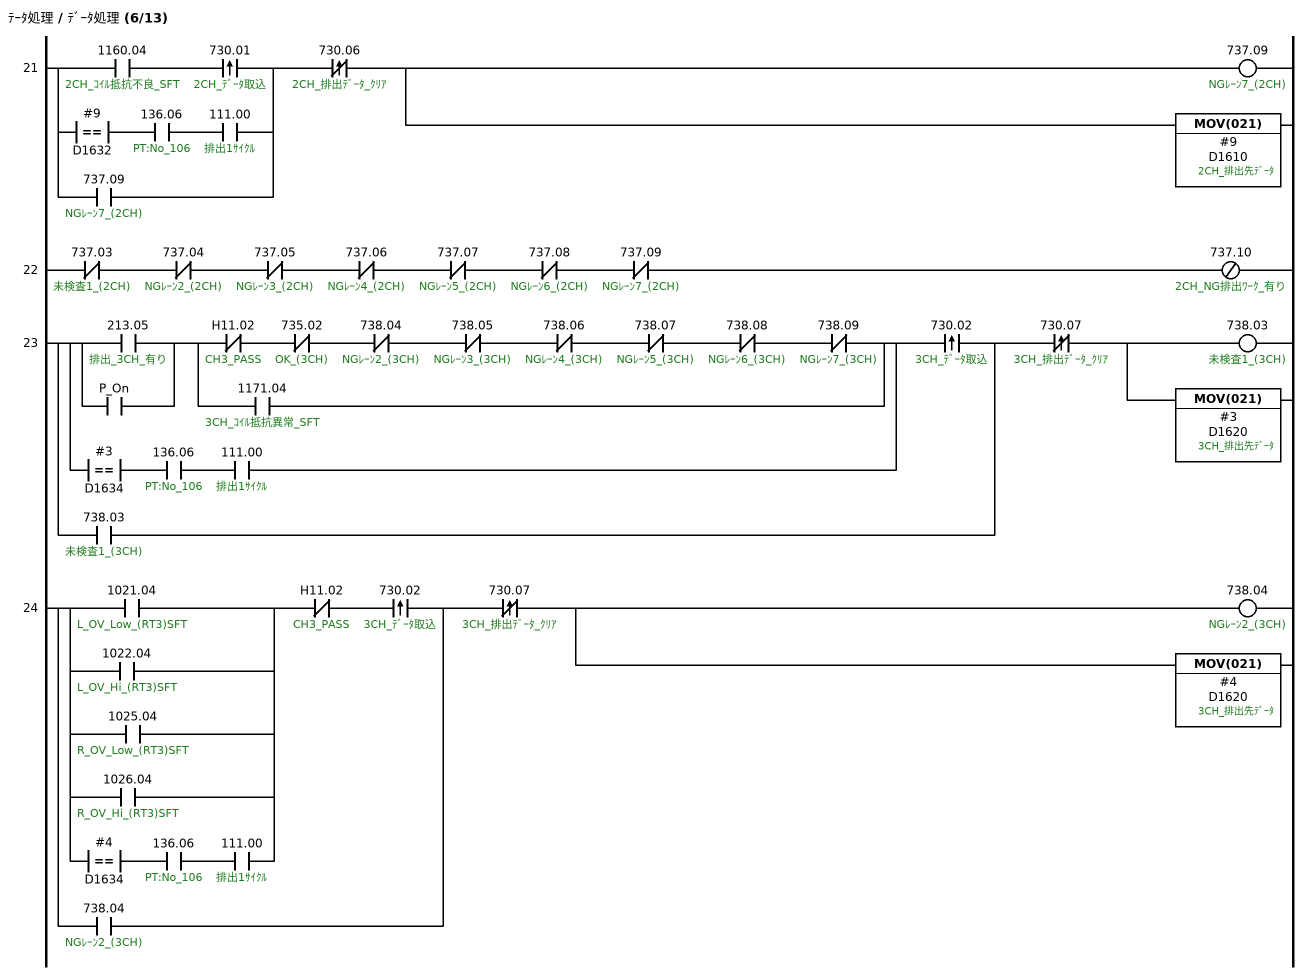
; [picture p168: ﾃｰﾀ処理 / ﾃﾞｰﾀ処理, rungs 21-24]
; rung 21
LD 1160.04  ; 2CH_ｺｲﾙ抵抗不良_SFT
@AND 730.01  ; 2CH_ﾃﾞｰﾀ取込
LD=(300) #9 D1632
AND 136.06  ; PT:No_106
AND 111.00  ; 排出1ｻｲｸﾙ
ORLD
OR 737.09  ; NGﾚｰﾝ7_(2CH)
@ANDNOT 730.06  ; 2CH_排出ﾃﾞｰﾀ_ｸﾘｱ
OUT 737.09  ; NGﾚｰﾝ7_(2CH)
MOV(021) #9 D1610  ; 2CH_排出先ﾃﾞｰﾀ
; rung 22
LDNOT 737.03  ; 未検査1_(2CH)
ANDNOT 737.04  ; NGﾚｰﾝ2_(2CH)
ANDNOT 737.05  ; NGﾚｰﾝ3_(2CH)
ANDNOT 737.06  ; NGﾚｰﾝ4_(2CH)
ANDNOT 737.07  ; NGﾚｰﾝ5_(2CH)
ANDNOT 737.08  ; NGﾚｰﾝ6_(2CH)
ANDNOT 737.09  ; NGﾚｰﾝ7_(2CH)
OUTNOT 737.10  ; 2CH_NG排出ﾜｰｸ_有り
; rung 23
LD 213.05  ; 排出_3CH_有り
OR P_On
LDNOT H11.02  ; CH3_PASS
ANDNOT 735.02  ; OK_(3CH)
ANDNOT 738.04  ; NGﾚｰﾝ2_(3CH)
ANDNOT 738.05  ; NGﾚｰﾝ3_(3CH)
ANDNOT 738.06  ; NGﾚｰﾝ4_(3CH)
ANDNOT 738.07  ; NGﾚｰﾝ5_(3CH)
ANDNOT 738.08  ; NGﾚｰﾝ6_(3CH)
ANDNOT 738.09  ; NGﾚｰﾝ7_(3CH)
OR 1171.04  ; 3CH_ｺｲﾙ抵抗異常_SFT
ANDLD
LD=(300) #3 D1634
AND 136.06  ; PT:No_106
AND 111.00  ; 排出1ｻｲｸﾙ
ORLD
@AND 730.02  ; 3CH_ﾃﾞｰﾀ取込
OR 738.03  ; 未検査1_(3CH)
@ANDNOT 730.07  ; 3CH_排出ﾃﾞｰﾀ_ｸﾘｱ
OUT 738.03  ; 未検査1_(3CH)
MOV(021) #3 D1620  ; 3CH_排出先ﾃﾞｰﾀ
; rung 24
LD 1021.04  ; L_OV_Low_(RT3)SFT
OR 1022.04  ; L_OV_Hi_(RT3)SFT
OR 1025.04  ; R_OV_Low_(RT3)SFT
OR 1026.04  ; R_OV_Hi_(RT3)SFT
LD=(300) #4 D1634
AND 136.06  ; PT:No_106
AND 111.00  ; 排出1ｻｲｸﾙ
ORLD
ANDNOT H11.02  ; CH3_PASS
@AND 730.02  ; 3CH_ﾃﾞｰﾀ取込
OR 738.04  ; NGﾚｰﾝ2_(3CH)
@ANDNOT 730.07  ; 3CH_排出ﾃﾞｰﾀ_ｸﾘｱ
OUT 738.04  ; NGﾚｰﾝ2_(3CH)
MOV(021) #4 D1620  ; 3CH_排出先ﾃﾞｰﾀ

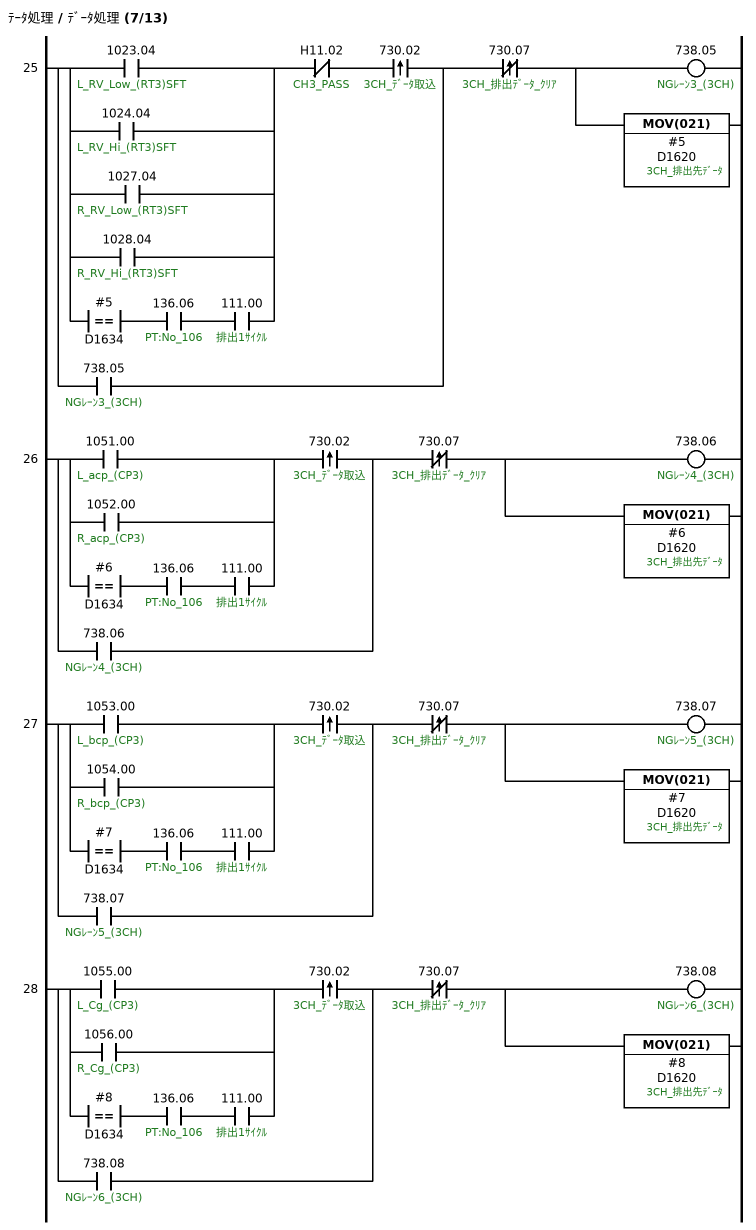
; rung 25
LD 1023.04  ; L_RV_Low_(RT3)SFT
OR 1024.04  ; L_RV_Hi_(RT3)SFT
OR 1027.04  ; R_RV_Low_(RT3)SFT
OR 1028.04  ; R_RV_Hi_(RT3)SFT
LD=(300) #5 D1634
AND 136.06  ; PT:No_106
AND 111.00  ; 排出1ｻｲｸﾙ
ORLD
ANDNOT H11.02  ; CH3_PASS
@AND 730.02  ; 3CH_ﾃﾞｰﾀ取込
OR 738.05  ; NGﾚｰﾝ3_(3CH)
@ANDNOT 730.07  ; 3CH_排出ﾃﾞｰﾀ_ｸﾘｱ
OUT 738.05  ; NGﾚｰﾝ3_(3CH)
MOV(021) #5 D1620  ; 3CH_排出先ﾃﾞｰﾀ
; rung 26
LD 1051.00  ; L_acp_(CP3)
OR 1052.00  ; R_acp_(CP3)
LD=(300) #6 D1634
AND 136.06  ; PT:No_106
AND 111.00  ; 排出1ｻｲｸﾙ
ORLD
@AND 730.02  ; 3CH_ﾃﾞｰﾀ取込
OR 738.06  ; NGﾚｰﾝ4_(3CH)
@ANDNOT 730.07  ; 3CH_排出ﾃﾞｰﾀ_ｸﾘｱ
OUT 738.06  ; NGﾚｰﾝ4_(3CH)
MOV(021) #6 D1620  ; 3CH_排出先ﾃﾞｰﾀ
; rung 27
LD 1053.00  ; L_bcp_(CP3)
OR 1054.00  ; R_bcp_(CP3)
LD=(300) #7 D1634
AND 136.06  ; PT:No_106
AND 111.00  ; 排出1ｻｲｸﾙ
ORLD
@AND 730.02  ; 3CH_ﾃﾞｰﾀ取込
OR 738.07  ; NGﾚｰﾝ5_(3CH)
@ANDNOT 730.07  ; 3CH_排出ﾃﾞｰﾀ_ｸﾘｱ
OUT 738.07  ; NGﾚｰﾝ5_(3CH)
MOV(021) #7 D1620  ; 3CH_排出先ﾃﾞｰﾀ
; rung 28
LD 1055.00  ; L_Cg_(CP3)
OR 1056.00  ; R_Cg_(CP3)
LD=(300) #8 D1634
AND 136.06  ; PT:No_106
AND 111.00  ; 排出1ｻｲｸﾙ
ORLD
@AND 730.02  ; 3CH_ﾃﾞｰﾀ取込
OR 738.08  ; NGﾚｰﾝ6_(3CH)
@ANDNOT 730.07  ; 3CH_排出ﾃﾞｰﾀ_ｸﾘｱ
OUT 738.08  ; NGﾚｰﾝ6_(3CH)
MOV(021) #8 D1620  ; 3CH_排出先ﾃﾞｰﾀ

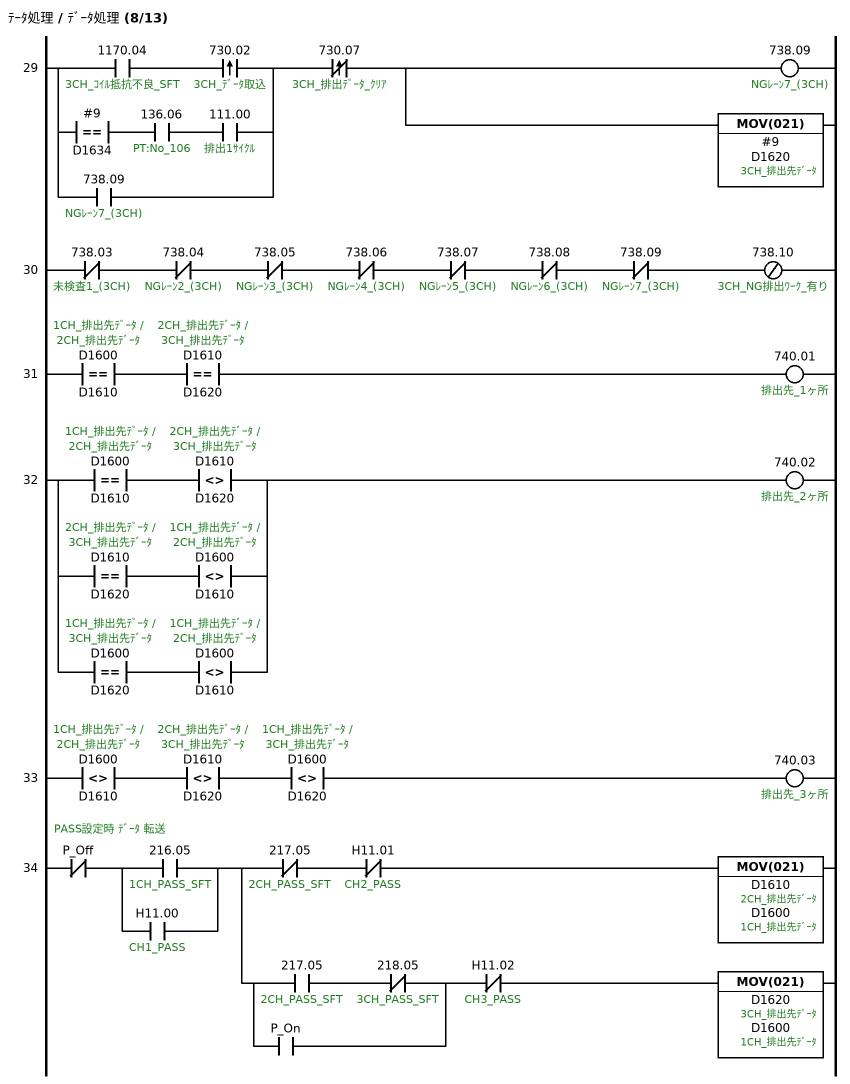
; rung 29
LD 1170.04  ; 3CH_ｺｲﾙ抵抗不良_SFT
@AND 730.02  ; 3CH_ﾃﾞｰﾀ取込
LD=(300) #9 D1634
AND 136.06  ; PT:No_106
AND 111.00  ; 排出1ｻｲｸﾙ
ORLD
OR 738.09  ; NGﾚｰﾝ7_(3CH)
@ANDNOT 730.07  ; 3CH_排出ﾃﾞｰﾀ_ｸﾘｱ
OUT 738.09  ; NGﾚｰﾝ7_(3CH)
MOV(021) #9 D1620  ; 3CH_排出先ﾃﾞｰﾀ
; rung 30
LDNOT 738.03  ; 未検査1_(3CH)
ANDNOT 738.04  ; NGﾚｰﾝ2_(3CH)
ANDNOT 738.05  ; NGﾚｰﾝ3_(3CH)
ANDNOT 738.06  ; NGﾚｰﾝ4_(3CH)
ANDNOT 738.07  ; NGﾚｰﾝ5_(3CH)
ANDNOT 738.08  ; NGﾚｰﾝ6_(3CH)
ANDNOT 738.09  ; NGﾚｰﾝ7_(3CH)
OUTNOT 738.10  ; 3CH_NG排出ﾜｰｸ_有り
; rung 31
LD=(300) D1600 D1610  ; 1CH_排出先ﾃﾞｰﾀ, 2CH_排出先ﾃﾞｰﾀ
AND=(300) D1610 D1620  ; 2CH_排出先ﾃﾞｰﾀ, 3CH_排出先ﾃﾞｰﾀ
OUT 740.01  ; 排出先_1ヶ所
; rung 32
LD=(300) D1600 D1610  ; 1CH_排出先ﾃﾞｰﾀ, 2CH_排出先ﾃﾞｰﾀ
AND<>(305) D1610 D1620  ; 2CH_排出先ﾃﾞｰﾀ, 3CH_排出先ﾃﾞｰﾀ
LD=(300) D1610 D1620  ; 2CH_排出先ﾃﾞｰﾀ, 3CH_排出先ﾃﾞｰﾀ
AND<>(305) D1600 D1610  ; 1CH_排出先ﾃﾞｰﾀ, 2CH_排出先ﾃﾞｰﾀ
ORLD
LD=(300) D1600 D1620  ; 1CH_排出先ﾃﾞｰﾀ, 3CH_排出先ﾃﾞｰﾀ
AND<>(305) D1600 D1610  ; 1CH_排出先ﾃﾞｰﾀ, 2CH_排出先ﾃﾞｰﾀ
ORLD
OUT 740.02  ; 排出先_2ヶ所
; rung 33
LD<>(305) D1600 D1610  ; 1CH_排出先ﾃﾞｰﾀ, 2CH_排出先ﾃﾞｰﾀ
AND<>(305) D1610 D1620  ; 2CH_排出先ﾃﾞｰﾀ, 3CH_排出先ﾃﾞｰﾀ
AND<>(305) D1600 D1620  ; 1CH_排出先ﾃﾞｰﾀ, 3CH_排出先ﾃﾞｰﾀ
OUT 740.03  ; 排出先_3ヶ所
; rung 34: PASS設定時 ﾃﾞｰﾀ 転送
LDNOT P_Off
LD 216.05  ; 1CH_PASS_SFT
OR H11.00  ; CH1_PASS
ANDLD
OUT TR0
ANDNOT 217.05  ; 2CH_PASS_SFT
ANDNOT H11.01  ; CH2_PASS
MOV(021) D1610 D1600  ; 2CH_排出先ﾃﾞｰﾀ, 1CH_排出先ﾃﾞｰﾀ
LD TR0
LD 217.05  ; 2CH_PASS_SFT
ANDNOT 218.05  ; 3CH_PASS_SFT
OR P_On
ANDLD
ANDNOT H11.02  ; CH3_PASS
MOV(021) D1620 D1600  ; 3CH_排出先ﾃﾞｰﾀ, 1CH_排出先ﾃﾞｰﾀ

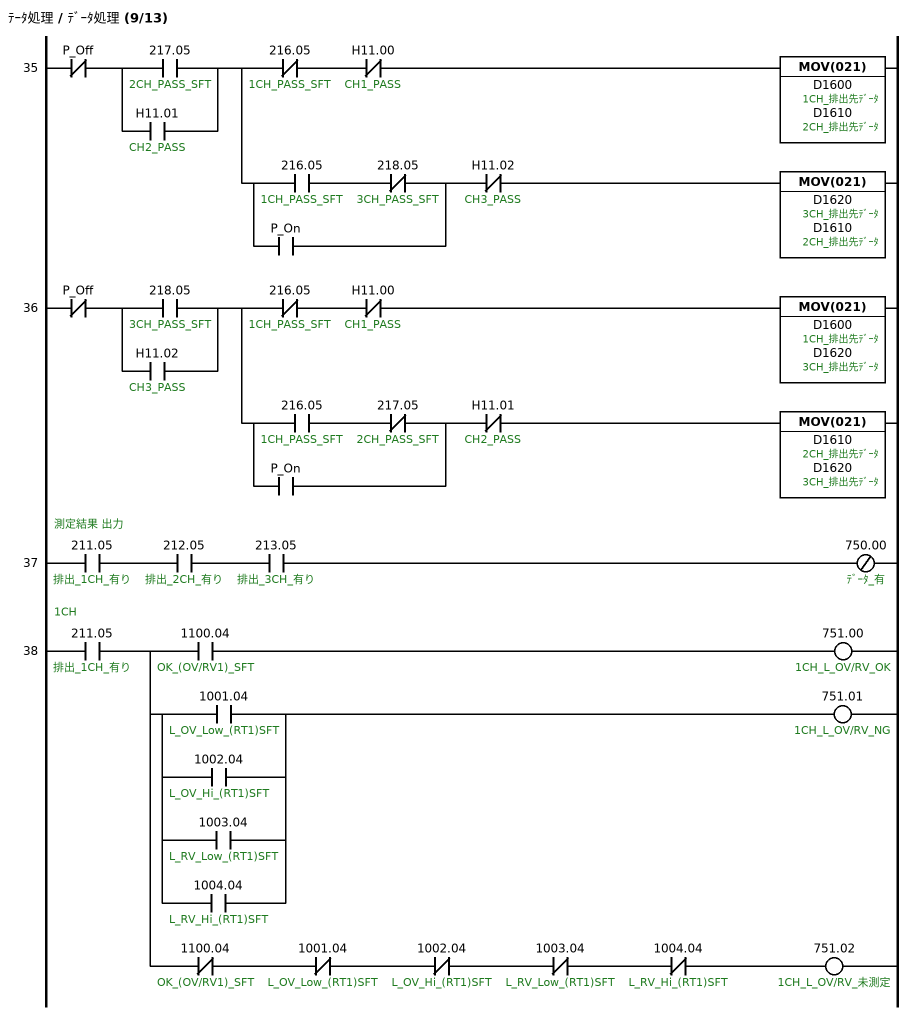
; rung 35
LDNOT P_Off
LD 217.05  ; 2CH_PASS_SFT
OR H11.01  ; CH2_PASS
ANDLD
OUT TR0
ANDNOT 216.05  ; 1CH_PASS_SFT
ANDNOT H11.00  ; CH1_PASS
MOV(021) D1600 D1610  ; 1CH_排出先ﾃﾞｰﾀ, 2CH_排出先ﾃﾞｰﾀ
LD TR0
LD 216.05  ; 1CH_PASS_SFT
ANDNOT 218.05  ; 3CH_PASS_SFT
OR P_On
ANDLD
ANDNOT H11.02  ; CH3_PASS
MOV(021) D1620 D1610  ; 3CH_排出先ﾃﾞｰﾀ, 2CH_排出先ﾃﾞｰﾀ
; rung 36
LDNOT P_Off
LD 218.05  ; 3CH_PASS_SFT
OR H11.02  ; CH3_PASS
ANDLD
OUT TR0
ANDNOT 216.05  ; 1CH_PASS_SFT
ANDNOT H11.00  ; CH1_PASS
MOV(021) D1600 D1620  ; 1CH_排出先ﾃﾞｰﾀ, 3CH_排出先ﾃﾞｰﾀ
LD TR0
LD 216.05  ; 1CH_PASS_SFT
ANDNOT 217.05  ; 2CH_PASS_SFT
OR P_On
ANDLD
ANDNOT H11.01  ; CH2_PASS
MOV(021) D1610 D1620  ; 2CH_排出先ﾃﾞｰﾀ, 3CH_排出先ﾃﾞｰﾀ
; rung 37: 測定結果 出力
LD 211.05  ; 排出_1CH_有り
AND 212.05  ; 排出_2CH_有り
AND 213.05  ; 排出_3CH_有り
OUTNOT 750.00  ; ﾃﾞｰﾀ_有
; rung 38: 1CH
LD 211.05  ; 排出_1CH_有り
OUT TR0
AND 1100.04  ; OK_(OV/RV1)_SFT
OUT 751.00  ; 1CH_L_OV/RV_OK
LD TR0
LD 1001.04  ; L_OV_Low_(RT1)SFT
OR 1002.04  ; L_OV_Hi_(RT1)SFT
OR 1003.04  ; L_RV_Low_(RT1)SFT
OR 1004.04  ; L_RV_Hi_(RT1)SFT
ANDLD
OUT 751.01  ; 1CH_L_OV/RV_NG
LD TR0
ANDNOT 1100.04  ; OK_(OV/RV1)_SFT
ANDNOT 1001.04  ; L_OV_Low_(RT1)SFT
ANDNOT 1002.04  ; L_OV_Hi_(RT1)SFT
ANDNOT 1003.04  ; L_RV_Low_(RT1)SFT
ANDNOT 1004.04  ; L_RV_Hi_(RT1)SFT
OUT 751.02  ; 1CH_L_OV/RV_未測定

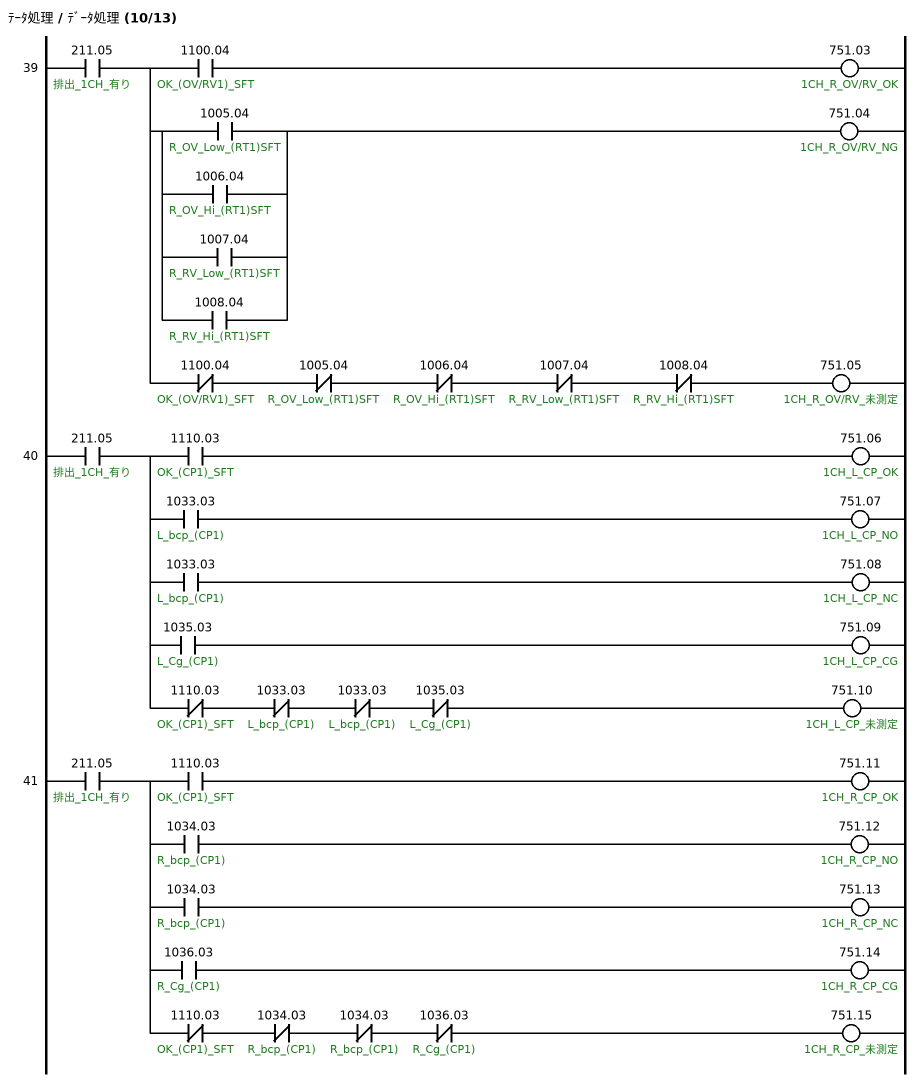
; rung 39
LD 211.05  ; 排出_1CH_有り
OUT TR0
AND 1100.04  ; OK_(OV/RV1)_SFT
OUT 751.03  ; 1CH_R_OV/RV_OK
LD TR0
LD 1005.04  ; R_OV_Low_(RT1)SFT
OR 1006.04  ; R_OV_Hi_(RT1)SFT
OR 1007.04  ; R_RV_Low_(RT1)SFT
OR 1008.04  ; R_RV_Hi_(RT1)SFT
ANDLD
OUT 751.04  ; 1CH_R_OV/RV_NG
LD TR0
ANDNOT 1100.04  ; OK_(OV/RV1)_SFT
ANDNOT 1005.04  ; R_OV_Low_(RT1)SFT
ANDNOT 1006.04  ; R_OV_Hi_(RT1)SFT
ANDNOT 1007.04  ; R_RV_Low_(RT1)SFT
ANDNOT 1008.04  ; R_RV_Hi_(RT1)SFT
OUT 751.05  ; 1CH_R_OV/RV_未測定
; rung 40
LD 211.05  ; 排出_1CH_有り
OUT TR0
AND 1110.03  ; OK_(CP1)_SFT
OUT 751.06  ; 1CH_L_CP_OK
LD TR0
AND 1033.03  ; L_bcp_(CP1)
OUT 751.07  ; 1CH_L_CP_NO
LD TR0
AND 1033.03  ; L_bcp_(CP1)
OUT 751.08  ; 1CH_L_CP_NC
LD TR0
AND 1035.03  ; L_Cg_(CP1)
OUT 751.09  ; 1CH_L_CP_CG
LD TR0
ANDNOT 1110.03  ; OK_(CP1)_SFT
ANDNOT 1033.03  ; L_bcp_(CP1)
ANDNOT 1033.03  ; L_bcp_(CP1)
ANDNOT 1035.03  ; L_Cg_(CP1)
OUT 751.10  ; 1CH_L_CP_未測定
; rung 41
LD 211.05  ; 排出_1CH_有り
OUT TR0
AND 1110.03  ; OK_(CP1)_SFT
OUT 751.11  ; 1CH_R_CP_OK
LD TR0
AND 1034.03  ; R_bcp_(CP1)
OUT 751.12  ; 1CH_R_CP_NO
LD TR0
AND 1034.03  ; R_bcp_(CP1)
OUT 751.13  ; 1CH_R_CP_NC
LD TR0
AND 1036.03  ; R_Cg_(CP1)
OUT 751.14  ; 1CH_R_CP_CG
LD TR0
ANDNOT 1110.03  ; OK_(CP1)_SFT
ANDNOT 1034.03  ; R_bcp_(CP1)
ANDNOT 1034.03  ; R_bcp_(CP1)
ANDNOT 1036.03  ; R_Cg_(CP1)
OUT 751.15  ; 1CH_R_CP_未測定

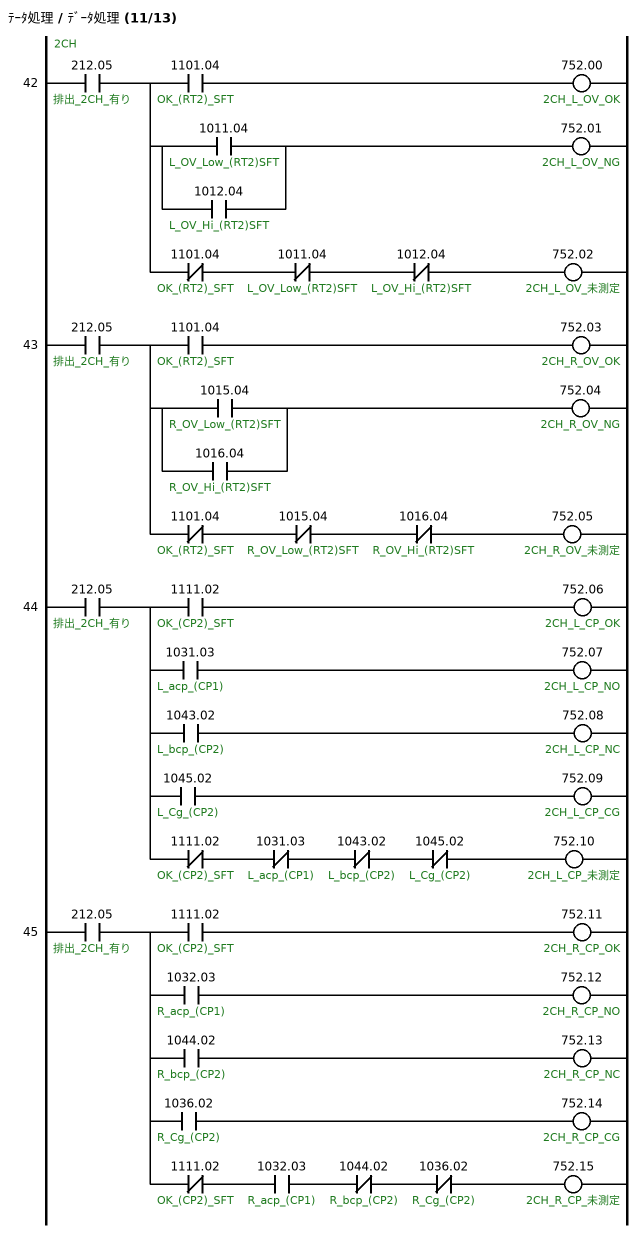
; rung 42: 2CH
LD 212.05  ; 排出_2CH_有り
OUT TR0
AND 1101.04  ; OK_(RT2)_SFT
OUT 752.00  ; 2CH_L_OV_OK
LD TR0
LD 1011.04  ; L_OV_Low_(RT2)SFT
OR 1012.04  ; L_OV_Hi_(RT2)SFT
ANDLD
OUT 752.01  ; 2CH_L_OV_NG
LD TR0
ANDNOT 1101.04  ; OK_(RT2)_SFT
ANDNOT 1011.04  ; L_OV_Low_(RT2)SFT
ANDNOT 1012.04  ; L_OV_Hi_(RT2)SFT
OUT 752.02  ; 2CH_L_OV_未測定
; rung 43
LD 212.05  ; 排出_2CH_有り
OUT TR0
AND 1101.04  ; OK_(RT2)_SFT
OUT 752.03  ; 2CH_R_OV_OK
LD TR0
LD 1015.04  ; R_OV_Low_(RT2)SFT
OR 1016.04  ; R_OV_Hi_(RT2)SFT
ANDLD
OUT 752.04  ; 2CH_R_OV_NG
LD TR0
ANDNOT 1101.04  ; OK_(RT2)_SFT
ANDNOT 1015.04  ; R_OV_Low_(RT2)SFT
ANDNOT 1016.04  ; R_OV_Hi_(RT2)SFT
OUT 752.05  ; 2CH_R_OV_未測定
; rung 44
LD 212.05  ; 排出_2CH_有り
OUT TR0
AND 1111.02  ; OK_(CP2)_SFT
OUT 752.06  ; 2CH_L_CP_OK
LD TR0
AND 1031.03  ; L_acp_(CP1)
OUT 752.07  ; 2CH_L_CP_NO
LD TR0
AND 1043.02  ; L_bcp_(CP2)
OUT 752.08  ; 2CH_L_CP_NC
LD TR0
AND 1045.02  ; L_Cg_(CP2)
OUT 752.09  ; 2CH_L_CP_CG
LD TR0
ANDNOT 1111.02  ; OK_(CP2)_SFT
ANDNOT 1031.03  ; L_acp_(CP1)
ANDNOT 1043.02  ; L_bcp_(CP2)
ANDNOT 1045.02  ; L_Cg_(CP2)
OUT 752.10  ; 2CH_L_CP_未測定
; rung 45
LD 212.05  ; 排出_2CH_有り
OUT TR0
AND 1111.02  ; OK_(CP2)_SFT
OUT 752.11  ; 2CH_R_CP_OK
LD TR0
AND 1032.03  ; R_acp_(CP1)
OUT 752.12  ; 2CH_R_CP_NO
LD TR0
AND 1044.02  ; R_bcp_(CP2)
OUT 752.13  ; 2CH_R_CP_NC
LD TR0
AND 1036.02  ; R_Cg_(CP2)
OUT 752.14  ; 2CH_R_CP_CG
LD TR0
ANDNOT 1111.02  ; OK_(CP2)_SFT
AND 1032.03  ; R_acp_(CP1)
ANDNOT 1044.02  ; R_bcp_(CP2)
ANDNOT 1036.02  ; R_Cg_(CP2)
OUT 752.15  ; 2CH_R_CP_未測定

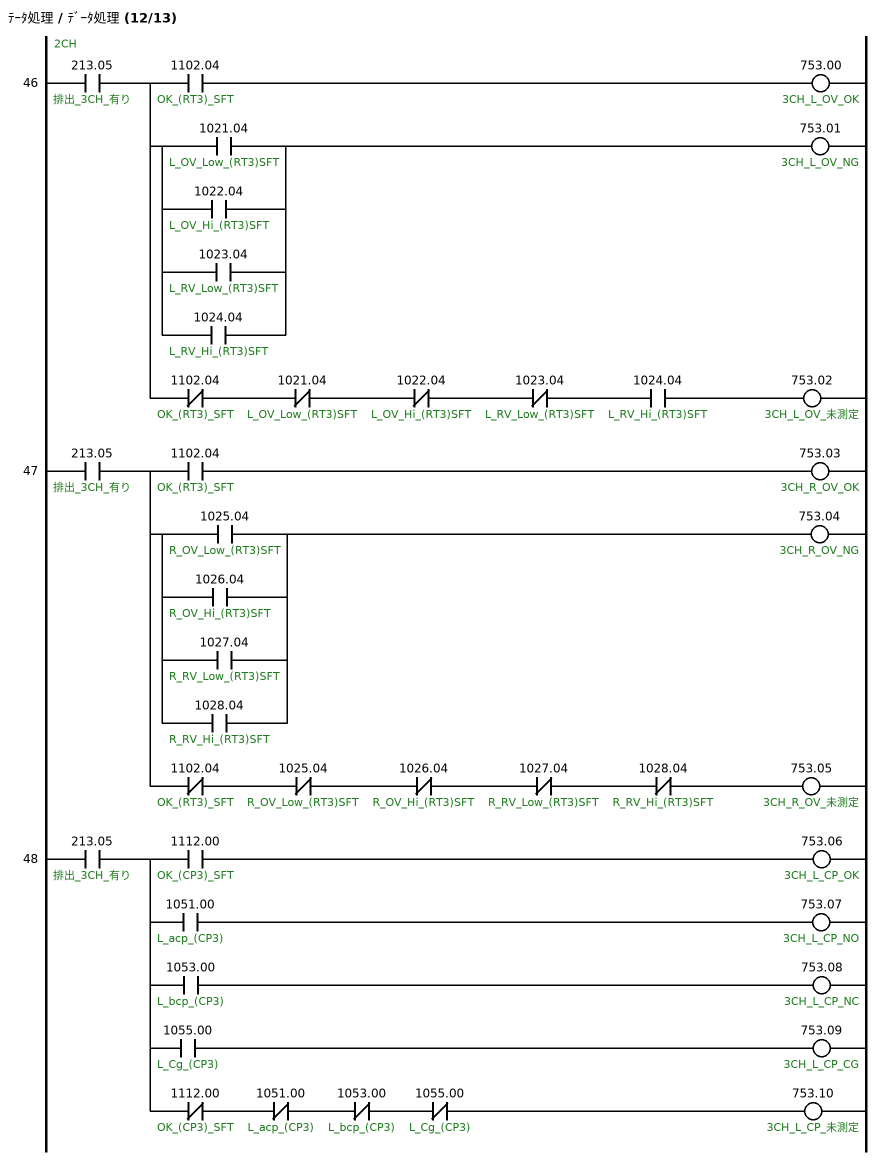
; rung 46: 2CH
LD 213.05  ; 排出_3CH_有り
OUT TR0
AND 1102.04  ; OK_(RT3)_SFT
OUT 753.00  ; 3CH_L_OV_OK
LD TR0
LD 1021.04  ; L_OV_Low_(RT3)SFT
OR 1022.04  ; L_OV_Hi_(RT3)SFT
OR 1023.04  ; L_RV_Low_(RT3)SFT
OR 1024.04  ; L_RV_Hi_(RT3)SFT
ANDLD
OUT 753.01  ; 3CH_L_OV_NG
LD TR0
ANDNOT 1102.04  ; OK_(RT3)_SFT
ANDNOT 1021.04  ; L_OV_Low_(RT3)SFT
ANDNOT 1022.04  ; L_OV_Hi_(RT3)SFT
ANDNOT 1023.04  ; L_RV_Low_(RT3)SFT
AND 1024.04  ; L_RV_Hi_(RT3)SFT
OUT 753.02  ; 3CH_L_OV_未測定
; rung 47
LD 213.05  ; 排出_3CH_有り
OUT TR0
AND 1102.04  ; OK_(RT3)_SFT
OUT 753.03  ; 3CH_R_OV_OK
LD TR0
LD 1025.04  ; R_OV_Low_(RT3)SFT
OR 1026.04  ; R_OV_Hi_(RT3)SFT
OR 1027.04  ; R_RV_Low_(RT3)SFT
OR 1028.04  ; R_RV_Hi_(RT3)SFT
ANDLD
OUT 753.04  ; 3CH_R_OV_NG
LD TR0
ANDNOT 1102.04  ; OK_(RT3)_SFT
ANDNOT 1025.04  ; R_OV_Low_(RT3)SFT
ANDNOT 1026.04  ; R_OV_Hi_(RT3)SFT
ANDNOT 1027.04  ; R_RV_Low_(RT3)SFT
ANDNOT 1028.04  ; R_RV_Hi_(RT3)SFT
OUT 753.05  ; 3CH_R_OV_未測定
; rung 48
LD 213.05  ; 排出_3CH_有り
OUT TR0
AND 1112.00  ; OK_(CP3)_SFT
OUT 753.06  ; 3CH_L_CP_OK
LD TR0
AND 1051.00  ; L_acp_(CP3)
OUT 753.07  ; 3CH_L_CP_NO
LD TR0
AND 1053.00  ; L_bcp_(CP3)
OUT 753.08  ; 3CH_L_CP_NC
LD TR0
AND 1055.00  ; L_Cg_(CP3)
OUT 753.09  ; 3CH_L_CP_CG
LD TR0
ANDNOT 1112.00  ; OK_(CP3)_SFT
ANDNOT 1051.00  ; L_acp_(CP3)
ANDNOT 1053.00  ; L_bcp_(CP3)
ANDNOT 1055.00  ; L_Cg_(CP3)
OUT 753.10  ; 3CH_L_CP_未測定

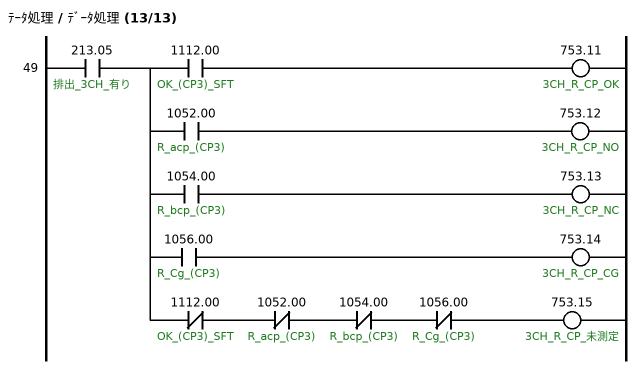
; rung 49
LD 213.05  ; 排出_3CH_有り
OUT TR0
AND 1112.00  ; OK_(CP3)_SFT
OUT 753.11  ; 3CH_R_CP_OK
LD TR0
AND 1052.00  ; R_acp_(CP3)
OUT 753.12  ; 3CH_R_CP_NO
LD TR0
AND 1054.00  ; R_bcp_(CP3)
OUT 753.13  ; 3CH_R_CP_NC
LD TR0
AND 1056.00  ; R_Cg_(CP3)
OUT 753.14  ; 3CH_R_CP_CG
LD TR0
ANDNOT 1112.00  ; OK_(CP3)_SFT
ANDNOT 1052.00  ; R_acp_(CP3)
ANDNOT 1054.00  ; R_bcp_(CP3)
ANDNOT 1056.00  ; R_Cg_(CP3)
OUT 753.15  ; 3CH_R_CP_未測定

### Section END
; rung 0
END(001)

## Program 排出 (cyclic task 7)

### Section 制御

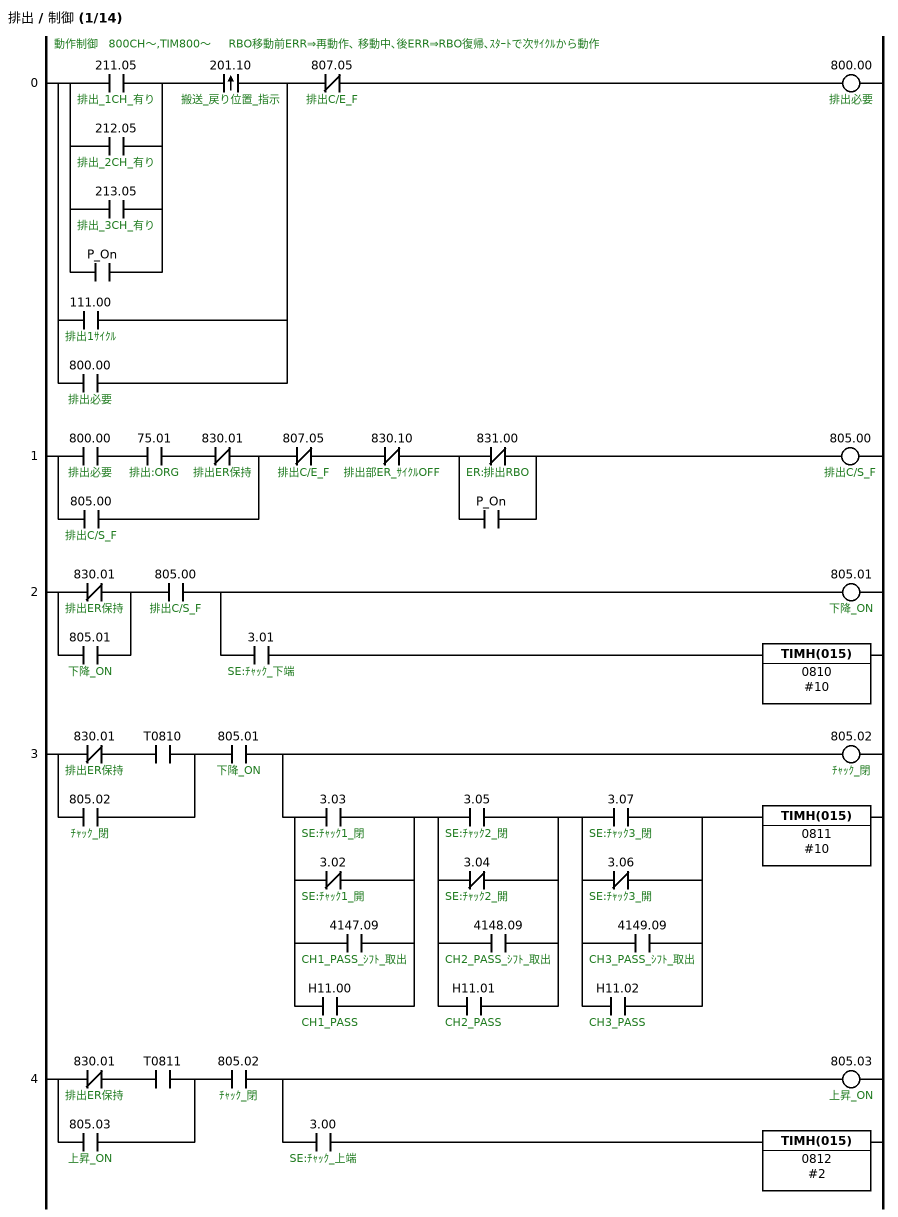
; rung 0: 動作制御   800CH～,TIM800～     RBO移動前ERR⇒再動作､ 移動中､後ERR⇒RBO復帰､ｽﾀｰﾄで次ｻｲｸﾙから動作
LD 211.05  ; 排出_1CH_有り
OR 212.05  ; 排出_2CH_有り
OR 213.05  ; 排出_3CH_有り
OR P_On
@AND 201.10  ; 搬送_戻り位置_指示
OR 111.00  ; 排出1ｻｲｸﾙ
OR 800.00  ; 排出必要
ANDNOT 807.05  ; 排出C/E_F
OUT 800.00  ; 排出必要
; rung 1
LD 800.00  ; 排出必要
AND 75.01  ; 排出:ORG
ANDNOT 830.01  ; 排出ER保持
OR 805.00  ; 排出C/S_F
ANDNOT 807.05  ; 排出C/E_F
ANDNOT 830.10  ; 排出部ER_ｻｲｸﾙOFF
LDNOT 831.00  ; ER:排出RBO
OR P_On
ANDLD
OUT 805.00  ; 排出C/S_F
; rung 2
LDNOT 830.01  ; 排出ER保持
OR 805.01  ; 下降_ON
AND 805.00  ; 排出C/S_F
OUT 805.01  ; 下降_ON
AND 3.01  ; SE:ﾁｬｯｸ_下端
TIMH(015) 0810 #10
; rung 3
LDNOT 830.01  ; 排出ER保持
AND T0810
OR 805.02  ; ﾁｬｯｸ_閉
AND 805.01  ; 下降_ON
OUT 805.02  ; ﾁｬｯｸ_閉
LD 3.03  ; SE:ﾁｬｯｸ1_閉
ORNOT 3.02  ; SE:ﾁｬｯｸ1_開
OR 4147.09  ; CH1_PASS_ｼﾌﾄ_取出
OR H11.00  ; CH1_PASS
ANDLD
LD 3.05  ; SE:ﾁｬｯｸ2_閉
ORNOT 3.04  ; SE:ﾁｬｯｸ2_開
OR 4148.09  ; CH2_PASS_ｼﾌﾄ_取出
OR H11.01  ; CH2_PASS
ANDLD
LD 3.07  ; SE:ﾁｬｯｸ3_閉
ORNOT 3.06  ; SE:ﾁｬｯｸ3_開
OR 4149.09  ; CH3_PASS_ｼﾌﾄ_取出
OR H11.02  ; CH3_PASS
ANDLD
TIMH(015) 0811 #10
; rung 4
LDNOT 830.01  ; 排出ER保持
AND T0811
OR 805.03  ; 上昇_ON
AND 805.02  ; ﾁｬｯｸ_閉
OUT 805.03  ; 上昇_ON
AND 3.00  ; SE:ﾁｬｯｸ_上端
TIMH(015) 0812 #2

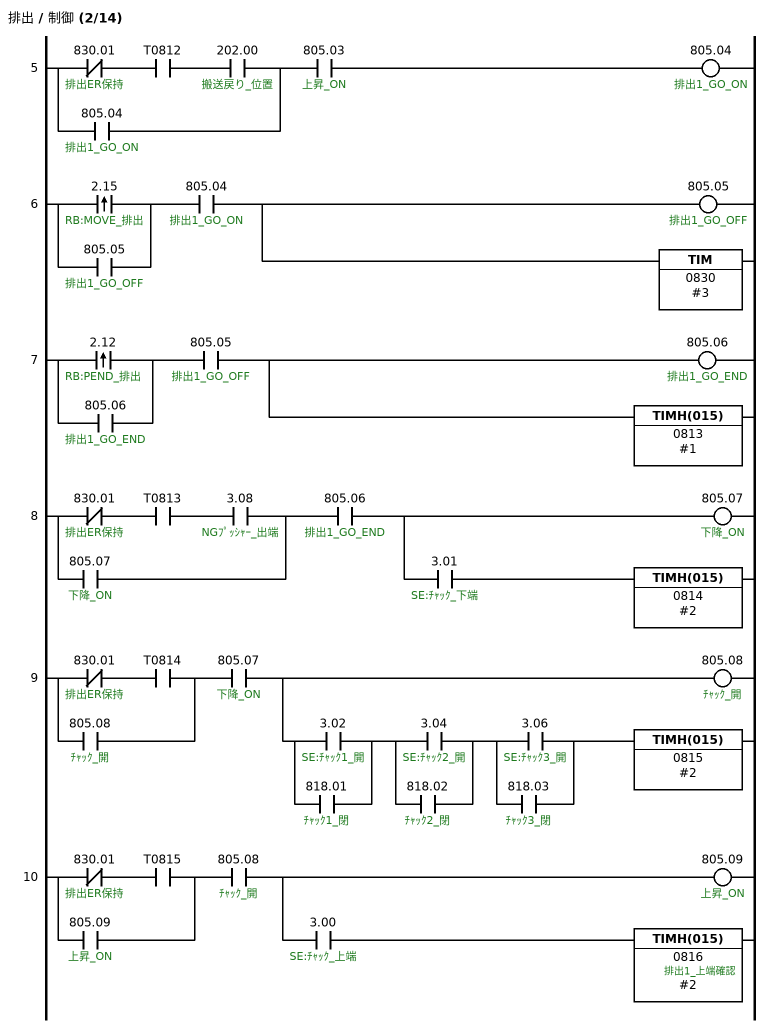
; rung 5
LDNOT 830.01  ; 排出ER保持
AND T0812
AND 202.00  ; 搬送戻り_位置
OR 805.04  ; 排出1_GO_ON
AND 805.03  ; 上昇_ON
OUT 805.04  ; 排出1_GO_ON
; rung 6
@LD 2.15  ; RB:MOVE_排出
OR 805.05  ; 排出1_GO_OFF
AND 805.04  ; 排出1_GO_ON
OUT 805.05  ; 排出1_GO_OFF
TIM 0830 #3
; rung 7
@LD 2.12  ; RB:PEND_排出
OR 805.06  ; 排出1_GO_END
AND 805.05  ; 排出1_GO_OFF
OUT 805.06  ; 排出1_GO_END
TIMH(015) 0813 #1
; rung 8
LDNOT 830.01  ; 排出ER保持
AND T0813
AND 3.08  ; NGﾌﾟｯｼｬｰ_出端
OR 805.07  ; 下降_ON
AND 805.06  ; 排出1_GO_END
OUT 805.07  ; 下降_ON
AND 3.01  ; SE:ﾁｬｯｸ_下端
TIMH(015) 0814 #2
; rung 9
LDNOT 830.01  ; 排出ER保持
AND T0814
OR 805.08  ; ﾁｬｯｸ_開
AND 805.07  ; 下降_ON
OUT 805.08  ; ﾁｬｯｸ_開
LD 3.02  ; SE:ﾁｬｯｸ1_開
OR 818.01  ; ﾁｬｯｸ1_閉
ANDLD
LD 3.04  ; SE:ﾁｬｯｸ2_開
OR 818.02  ; ﾁｬｯｸ2_閉
ANDLD
LD 3.06  ; SE:ﾁｬｯｸ3_開
OR 818.03  ; ﾁｬｯｸ3_閉
ANDLD
TIMH(015) 0815 #2
; rung 10
LDNOT 830.01  ; 排出ER保持
AND T0815
OR 805.09  ; 上昇_ON
AND 805.08  ; ﾁｬｯｸ_開
OUT 805.09  ; 上昇_ON
AND 3.00  ; SE:ﾁｬｯｸ_上端
TIMH(015) 0816 #2  ; 排出1_上端確認

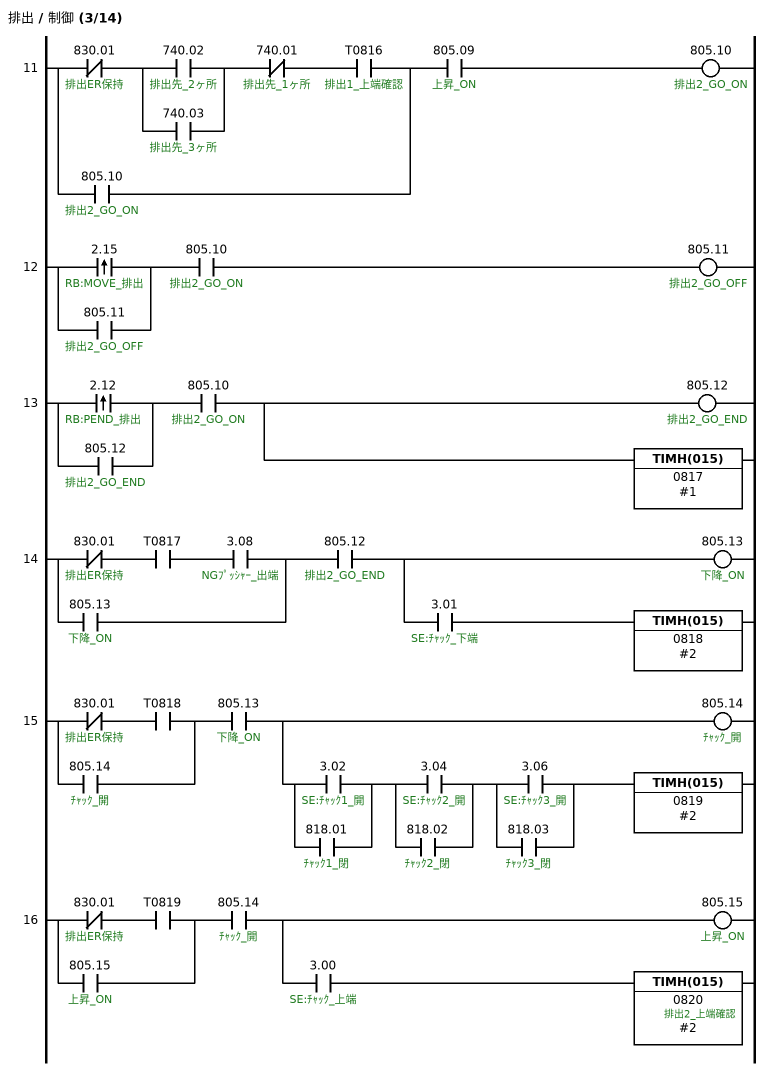
; rung 11
LDNOT 830.01  ; 排出ER保持
LD 740.02  ; 排出先_2ヶ所
OR 740.03  ; 排出先_3ヶ所
ANDLD
ANDNOT 740.01  ; 排出先_1ヶ所
AND T0816  ; 排出1_上端確認
OR 805.10  ; 排出2_GO_ON
AND 805.09  ; 上昇_ON
OUT 805.10  ; 排出2_GO_ON
; rung 12
@LD 2.15  ; RB:MOVE_排出
OR 805.11  ; 排出2_GO_OFF
AND 805.10  ; 排出2_GO_ON
OUT 805.11  ; 排出2_GO_OFF
; rung 13
@LD 2.12  ; RB:PEND_排出
OR 805.12  ; 排出2_GO_END
AND 805.10  ; 排出2_GO_ON
OUT 805.12  ; 排出2_GO_END
TIMH(015) 0817 #1
; rung 14
LDNOT 830.01  ; 排出ER保持
AND T0817
AND 3.08  ; NGﾌﾟｯｼｬｰ_出端
OR 805.13  ; 下降_ON
AND 805.12  ; 排出2_GO_END
OUT 805.13  ; 下降_ON
AND 3.01  ; SE:ﾁｬｯｸ_下端
TIMH(015) 0818 #2
; rung 15
LDNOT 830.01  ; 排出ER保持
AND T0818
OR 805.14  ; ﾁｬｯｸ_開
AND 805.13  ; 下降_ON
OUT 805.14  ; ﾁｬｯｸ_開
LD 3.02  ; SE:ﾁｬｯｸ1_開
OR 818.01  ; ﾁｬｯｸ1_閉
ANDLD
LD 3.04  ; SE:ﾁｬｯｸ2_開
OR 818.02  ; ﾁｬｯｸ2_閉
ANDLD
LD 3.06  ; SE:ﾁｬｯｸ3_開
OR 818.03  ; ﾁｬｯｸ3_閉
ANDLD
TIMH(015) 0819 #2
; rung 16
LDNOT 830.01  ; 排出ER保持
AND T0819
OR 805.15  ; 上昇_ON
AND 805.14  ; ﾁｬｯｸ_開
OUT 805.15  ; 上昇_ON
AND 3.00  ; SE:ﾁｬｯｸ_上端
TIMH(015) 0820 #2  ; 排出2_上端確認

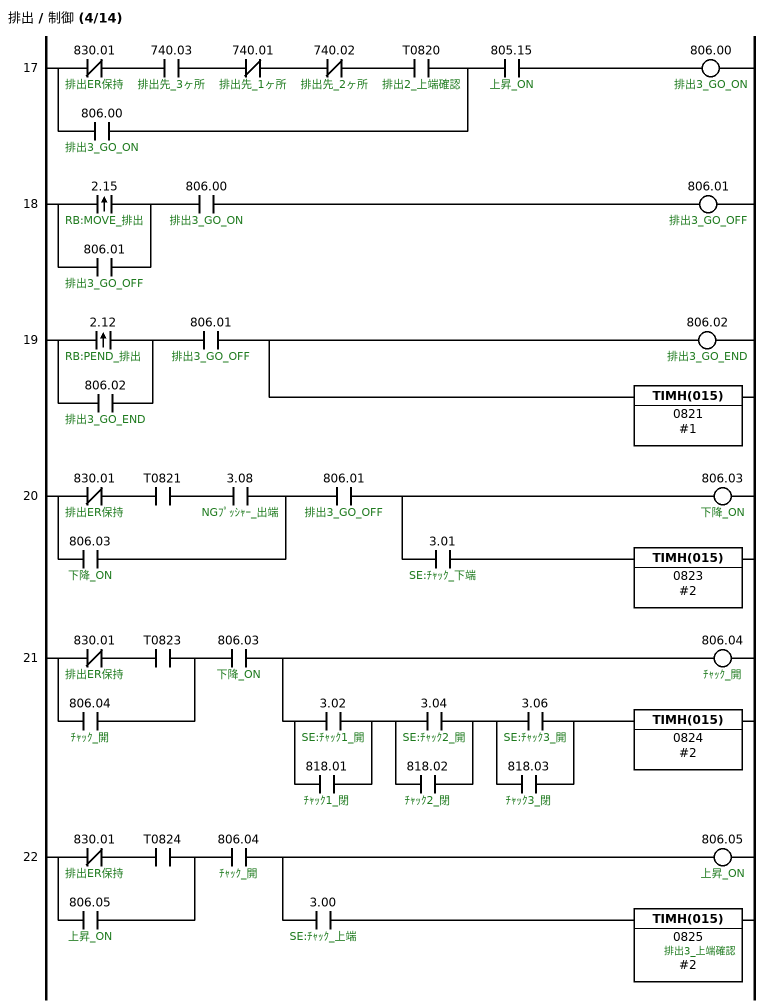
; rung 17
LDNOT 830.01  ; 排出ER保持
AND 740.03  ; 排出先_3ヶ所
ANDNOT 740.01  ; 排出先_1ヶ所
ANDNOT 740.02  ; 排出先_2ヶ所
AND T0820  ; 排出2_上端確認
OR 806.00  ; 排出3_GO_ON
AND 805.15  ; 上昇_ON
OUT 806.00  ; 排出3_GO_ON
; rung 18
@LD 2.15  ; RB:MOVE_排出
OR 806.01  ; 排出3_GO_OFF
AND 806.00  ; 排出3_GO_ON
OUT 806.01  ; 排出3_GO_OFF
; rung 19
@LD 2.12  ; RB:PEND_排出
OR 806.02  ; 排出3_GO_END
AND 806.01  ; 排出3_GO_OFF
OUT 806.02  ; 排出3_GO_END
TIMH(015) 0821 #1
; rung 20
LDNOT 830.01  ; 排出ER保持
AND T0821
AND 3.08  ; NGﾌﾟｯｼｬｰ_出端
OR 806.03  ; 下降_ON
AND 806.01  ; 排出3_GO_OFF
OUT 806.03  ; 下降_ON
AND 3.01  ; SE:ﾁｬｯｸ_下端
TIMH(015) 0823 #2
; rung 21
LDNOT 830.01  ; 排出ER保持
AND T0823
OR 806.04  ; ﾁｬｯｸ_開
AND 806.03  ; 下降_ON
OUT 806.04  ; ﾁｬｯｸ_開
LD 3.02  ; SE:ﾁｬｯｸ1_開
OR 818.01  ; ﾁｬｯｸ1_閉
ANDLD
LD 3.04  ; SE:ﾁｬｯｸ2_開
OR 818.02  ; ﾁｬｯｸ2_閉
ANDLD
LD 3.06  ; SE:ﾁｬｯｸ3_開
OR 818.03  ; ﾁｬｯｸ3_閉
ANDLD
TIMH(015) 0824 #2
; rung 22
LDNOT 830.01  ; 排出ER保持
AND T0824
OR 806.05  ; 上昇_ON
AND 806.04  ; ﾁｬｯｸ_開
OUT 806.05  ; 上昇_ON
AND 3.00  ; SE:ﾁｬｯｸ_上端
TIMH(015) 0825 #2  ; 排出3_上端確認

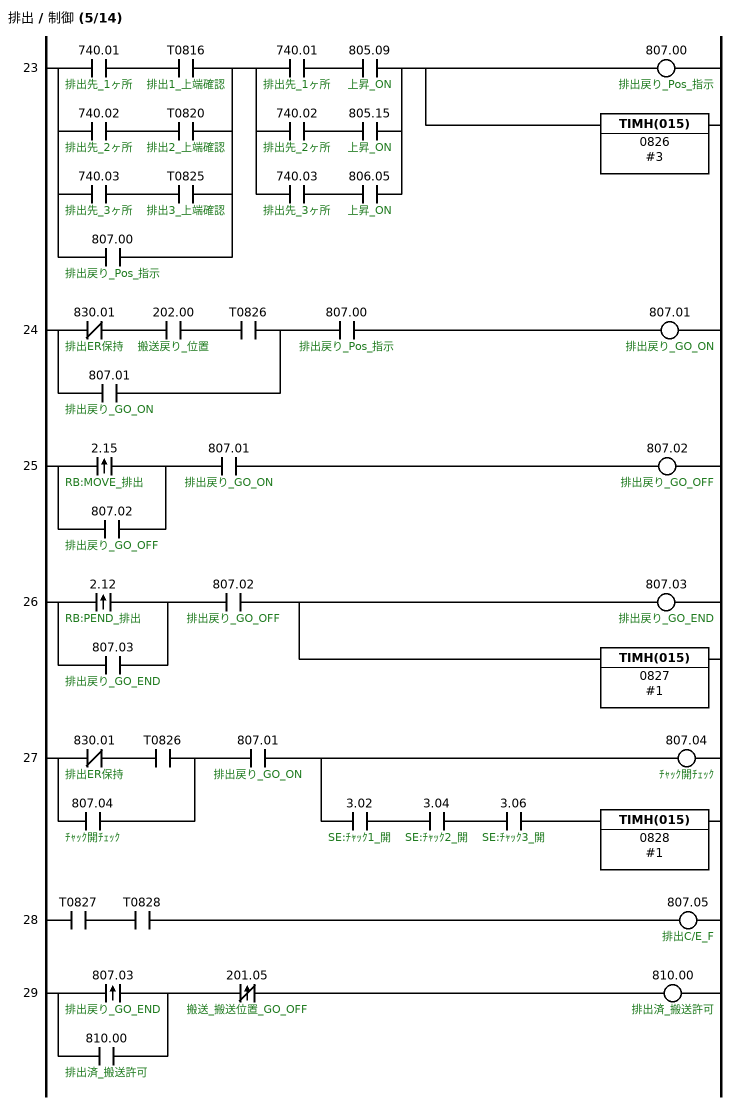
; rung 23
LD 740.01  ; 排出先_1ヶ所
AND T0816  ; 排出1_上端確認
LD 740.02  ; 排出先_2ヶ所
AND T0820  ; 排出2_上端確認
ORLD
LD 740.03  ; 排出先_3ヶ所
AND T0825  ; 排出3_上端確認
ORLD
OR 807.00  ; 排出戻り_Pos_指示
LD 740.01  ; 排出先_1ヶ所
AND 805.09  ; 上昇_ON
LD 740.02  ; 排出先_2ヶ所
AND 805.15  ; 上昇_ON
ORLD
LD 740.03  ; 排出先_3ヶ所
AND 806.05  ; 上昇_ON
ORLD
ANDLD
OUT 807.00  ; 排出戻り_Pos_指示
TIMH(015) 0826 #3
; rung 24
LDNOT 830.01  ; 排出ER保持
AND 202.00  ; 搬送戻り_位置
AND T0826
OR 807.01  ; 排出戻り_GO_ON
AND 807.00  ; 排出戻り_Pos_指示
OUT 807.01  ; 排出戻り_GO_ON
; rung 25
@LD 2.15  ; RB:MOVE_排出
OR 807.02  ; 排出戻り_GO_OFF
AND 807.01  ; 排出戻り_GO_ON
OUT 807.02  ; 排出戻り_GO_OFF
; rung 26
@LD 2.12  ; RB:PEND_排出
OR 807.03  ; 排出戻り_GO_END
AND 807.02  ; 排出戻り_GO_OFF
OUT 807.03  ; 排出戻り_GO_END
TIMH(015) 0827 #1
; rung 27
LDNOT 830.01  ; 排出ER保持
AND T0826
OR 807.04  ; ﾁｬｯｸ開ﾁｪｯｸ
AND 807.01  ; 排出戻り_GO_ON
OUT 807.04  ; ﾁｬｯｸ開ﾁｪｯｸ
AND 3.02  ; SE:ﾁｬｯｸ1_開
AND 3.04  ; SE:ﾁｬｯｸ2_開
AND 3.06  ; SE:ﾁｬｯｸ3_開
TIMH(015) 0828 #1
; rung 28
LD T0827
AND T0828
OUT 807.05  ; 排出C/E_F
; rung 29
@LD 807.03  ; 排出戻り_GO_END
OR 810.00  ; 排出済_搬送許可
@ANDNOT 201.05  ; 搬送_搬送位置_GO_OFF
OUT 810.00  ; 排出済_搬送許可

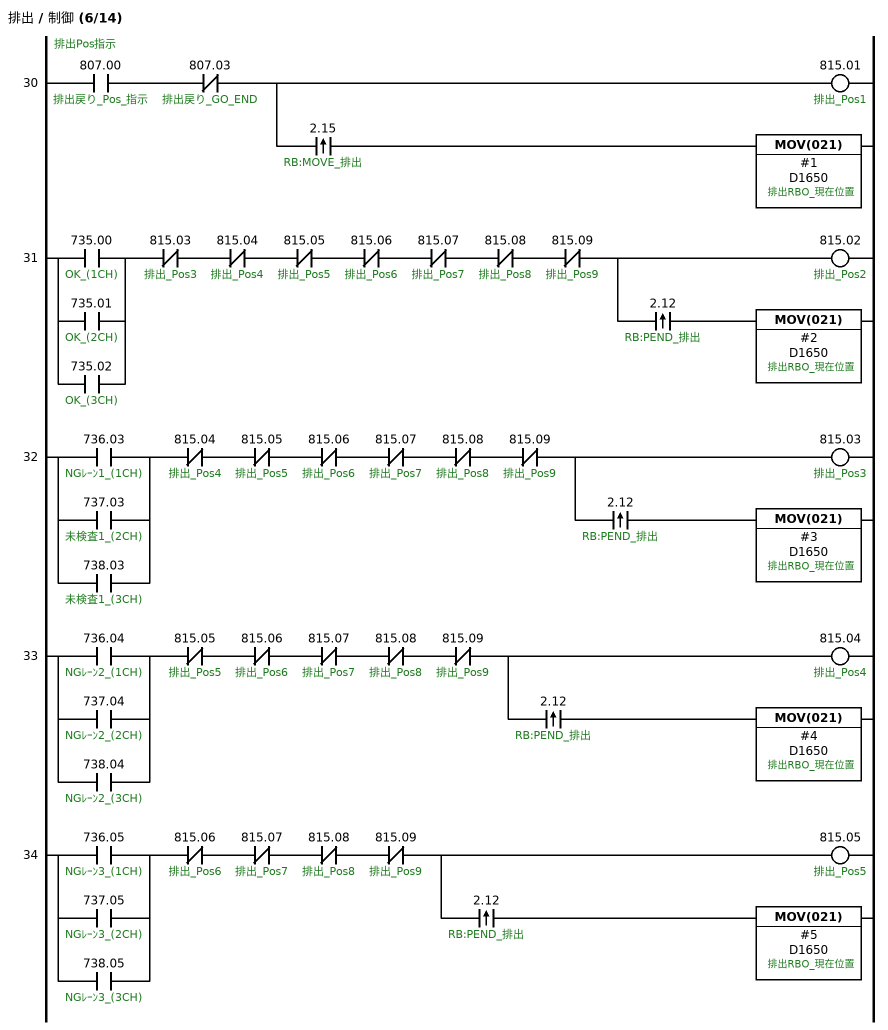
; rung 30: 排出Pos指示
LD 807.00  ; 排出戻り_Pos_指示
ANDNOT 807.03  ; 排出戻り_GO_END
OUT 815.01  ; 排出_Pos1
@AND 2.15  ; RB:MOVE_排出
MOV(021) #1 D1650  ; 排出RBO_現在位置
; rung 31
LD 735.00  ; OK_(1CH)
OR 735.01  ; OK_(2CH)
OR 735.02  ; OK_(3CH)
ANDNOT 815.03  ; 排出_Pos3
ANDNOT 815.04  ; 排出_Pos4
ANDNOT 815.05  ; 排出_Pos5
ANDNOT 815.06  ; 排出_Pos6
ANDNOT 815.07  ; 排出_Pos7
ANDNOT 815.08  ; 排出_Pos8
ANDNOT 815.09  ; 排出_Pos9
OUT 815.02  ; 排出_Pos2
@AND 2.12  ; RB:PEND_排出
MOV(021) #2 D1650  ; 排出RBO_現在位置
; rung 32
LD 736.03  ; NGﾚｰﾝ1_(1CH)
OR 737.03  ; 未検査1_(2CH)
OR 738.03  ; 未検査1_(3CH)
ANDNOT 815.04  ; 排出_Pos4
ANDNOT 815.05  ; 排出_Pos5
ANDNOT 815.06  ; 排出_Pos6
ANDNOT 815.07  ; 排出_Pos7
ANDNOT 815.08  ; 排出_Pos8
ANDNOT 815.09  ; 排出_Pos9
OUT 815.03  ; 排出_Pos3
@AND 2.12  ; RB:PEND_排出
MOV(021) #3 D1650  ; 排出RBO_現在位置
; rung 33
LD 736.04  ; NGﾚｰﾝ2_(1CH)
OR 737.04  ; NGﾚｰﾝ2_(2CH)
OR 738.04  ; NGﾚｰﾝ2_(3CH)
ANDNOT 815.05  ; 排出_Pos5
ANDNOT 815.06  ; 排出_Pos6
ANDNOT 815.07  ; 排出_Pos7
ANDNOT 815.08  ; 排出_Pos8
ANDNOT 815.09  ; 排出_Pos9
OUT 815.04  ; 排出_Pos4
@AND 2.12  ; RB:PEND_排出
MOV(021) #4 D1650  ; 排出RBO_現在位置
; rung 34
LD 736.05  ; NGﾚｰﾝ3_(1CH)
OR 737.05  ; NGﾚｰﾝ3_(2CH)
OR 738.05  ; NGﾚｰﾝ3_(3CH)
ANDNOT 815.06  ; 排出_Pos6
ANDNOT 815.07  ; 排出_Pos7
ANDNOT 815.08  ; 排出_Pos8
ANDNOT 815.09  ; 排出_Pos9
OUT 815.05  ; 排出_Pos5
@AND 2.12  ; RB:PEND_排出
MOV(021) #5 D1650  ; 排出RBO_現在位置

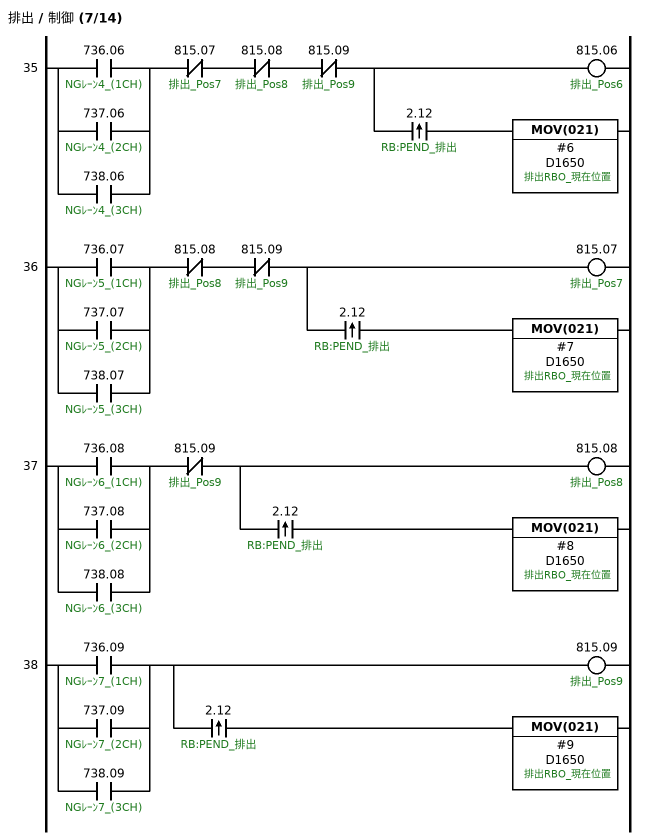
; rung 35
LD 736.06  ; NGﾚｰﾝ4_(1CH)
OR 737.06  ; NGﾚｰﾝ4_(2CH)
OR 738.06  ; NGﾚｰﾝ4_(3CH)
ANDNOT 815.07  ; 排出_Pos7
ANDNOT 815.08  ; 排出_Pos8
ANDNOT 815.09  ; 排出_Pos9
OUT 815.06  ; 排出_Pos6
@AND 2.12  ; RB:PEND_排出
MOV(021) #6 D1650  ; 排出RBO_現在位置
; rung 36
LD 736.07  ; NGﾚｰﾝ5_(1CH)
OR 737.07  ; NGﾚｰﾝ5_(2CH)
OR 738.07  ; NGﾚｰﾝ5_(3CH)
ANDNOT 815.08  ; 排出_Pos8
ANDNOT 815.09  ; 排出_Pos9
OUT 815.07  ; 排出_Pos7
@AND 2.12  ; RB:PEND_排出
MOV(021) #7 D1650  ; 排出RBO_現在位置
; rung 37
LD 736.08  ; NGﾚｰﾝ6_(1CH)
OR 737.08  ; NGﾚｰﾝ6_(2CH)
OR 738.08  ; NGﾚｰﾝ6_(3CH)
ANDNOT 815.09  ; 排出_Pos9
OUT 815.08  ; 排出_Pos8
@AND 2.12  ; RB:PEND_排出
MOV(021) #8 D1650  ; 排出RBO_現在位置
; rung 38
LD 736.09  ; NGﾚｰﾝ7_(1CH)
OR 737.09  ; NGﾚｰﾝ7_(2CH)
OR 738.09  ; NGﾚｰﾝ7_(3CH)
OUT 815.09  ; 排出_Pos9
@AND 2.12  ; RB:PEND_排出
MOV(021) #9 D1650  ; 排出RBO_現在位置

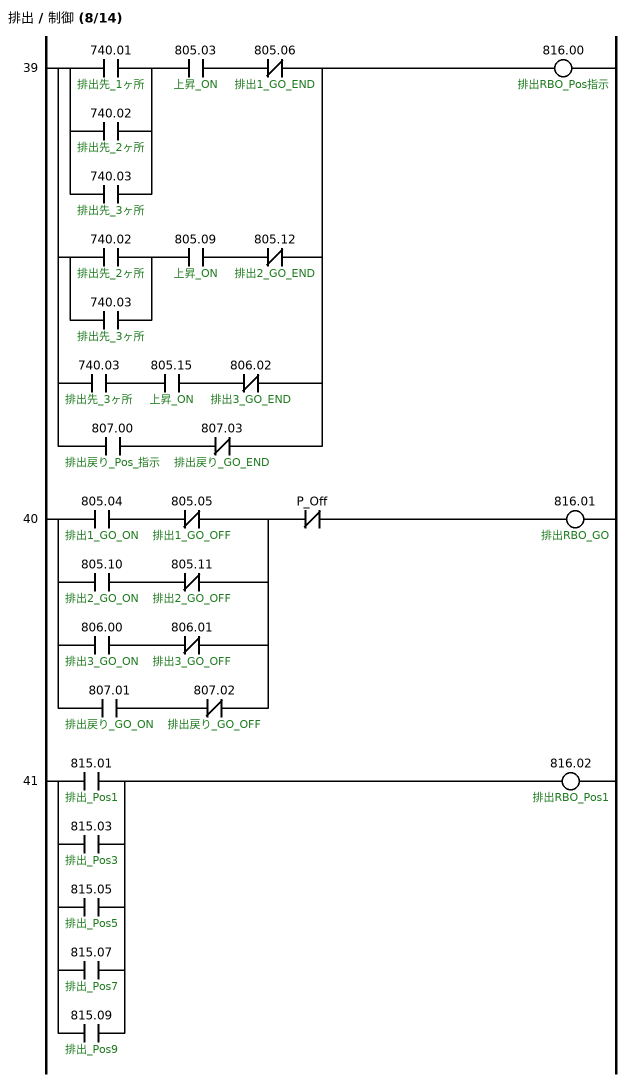
; rung 39
LD 740.01  ; 排出先_1ヶ所
OR 740.02  ; 排出先_2ヶ所
OR 740.03  ; 排出先_3ヶ所
AND 805.03  ; 上昇_ON
ANDNOT 805.06  ; 排出1_GO_END
LD 740.02  ; 排出先_2ヶ所
OR 740.03  ; 排出先_3ヶ所
AND 805.09  ; 上昇_ON
ANDNOT 805.12  ; 排出2_GO_END
ORLD
LD 740.03  ; 排出先_3ヶ所
AND 805.15  ; 上昇_ON
ANDNOT 806.02  ; 排出3_GO_END
ORLD
LD 807.00  ; 排出戻り_Pos_指示
ANDNOT 807.03  ; 排出戻り_GO_END
ORLD
OUT 816.00  ; 排出RBO_Pos指示
; rung 40
LD 805.04  ; 排出1_GO_ON
ANDNOT 805.05  ; 排出1_GO_OFF
LD 805.10  ; 排出2_GO_ON
ANDNOT 805.11  ; 排出2_GO_OFF
ORLD
LD 806.00  ; 排出3_GO_ON
ANDNOT 806.01  ; 排出3_GO_OFF
ORLD
LD 807.01  ; 排出戻り_GO_ON
ANDNOT 807.02  ; 排出戻り_GO_OFF
ORLD
ANDNOT P_Off
OUT 816.01  ; 排出RBO_GO
; rung 41
LD 815.01  ; 排出_Pos1
OR 815.03  ; 排出_Pos3
OR 815.05  ; 排出_Pos5
OR 815.07  ; 排出_Pos7
OR 815.09  ; 排出_Pos9
OUT 816.02  ; 排出RBO_Pos1

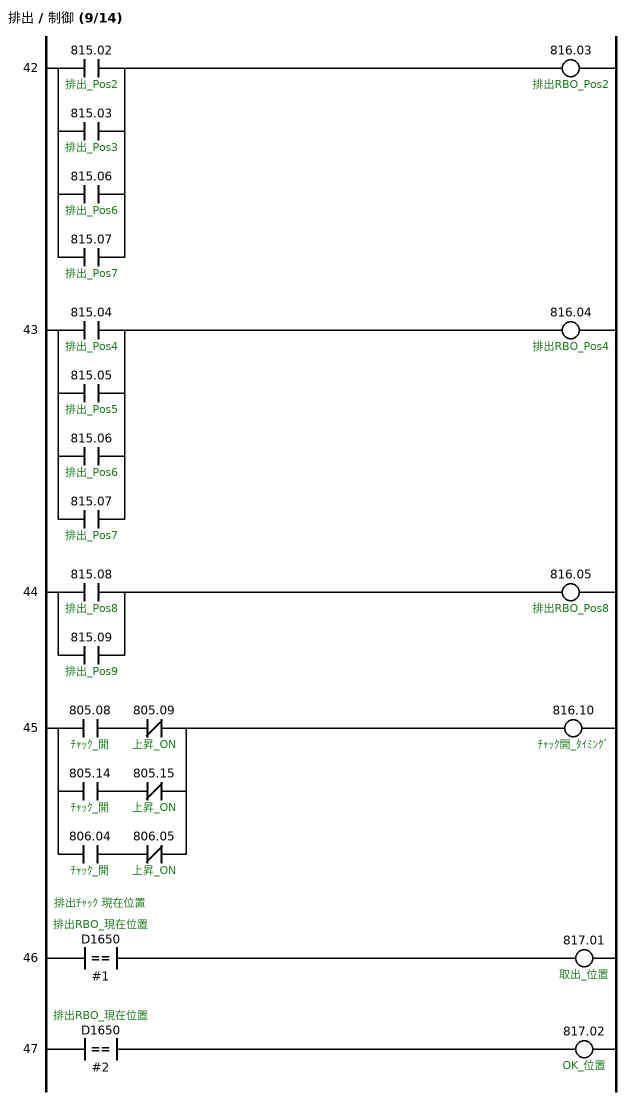
; rung 42
LD 815.02  ; 排出_Pos2
OR 815.03  ; 排出_Pos3
OR 815.06  ; 排出_Pos6
OR 815.07  ; 排出_Pos7
OUT 816.03  ; 排出RBO_Pos2
; rung 43
LD 815.04  ; 排出_Pos4
OR 815.05  ; 排出_Pos5
OR 815.06  ; 排出_Pos6
OR 815.07  ; 排出_Pos7
OUT 816.04  ; 排出RBO_Pos4
; rung 44
LD 815.08  ; 排出_Pos8
OR 815.09  ; 排出_Pos9
OUT 816.05  ; 排出RBO_Pos8
; rung 45
LD 805.08  ; ﾁｬｯｸ_開
ANDNOT 805.09  ; 上昇_ON
LD 805.14  ; ﾁｬｯｸ_開
ANDNOT 805.15  ; 上昇_ON
ORLD
LD 806.04  ; ﾁｬｯｸ_開
ANDNOT 806.05  ; 上昇_ON
ORLD
OUT 816.10  ; ﾁｬｯｸ開_ﾀｲﾐﾝｸﾞ
; rung 46: 排出ﾁｬｯｸ 現在位置
LD=(300) D1650 #1  ; 排出RBO_現在位置
OUT 817.01  ; 取出_位置
; rung 47
LD=(300) D1650 #2  ; 排出RBO_現在位置
OUT 817.02  ; OK_位置

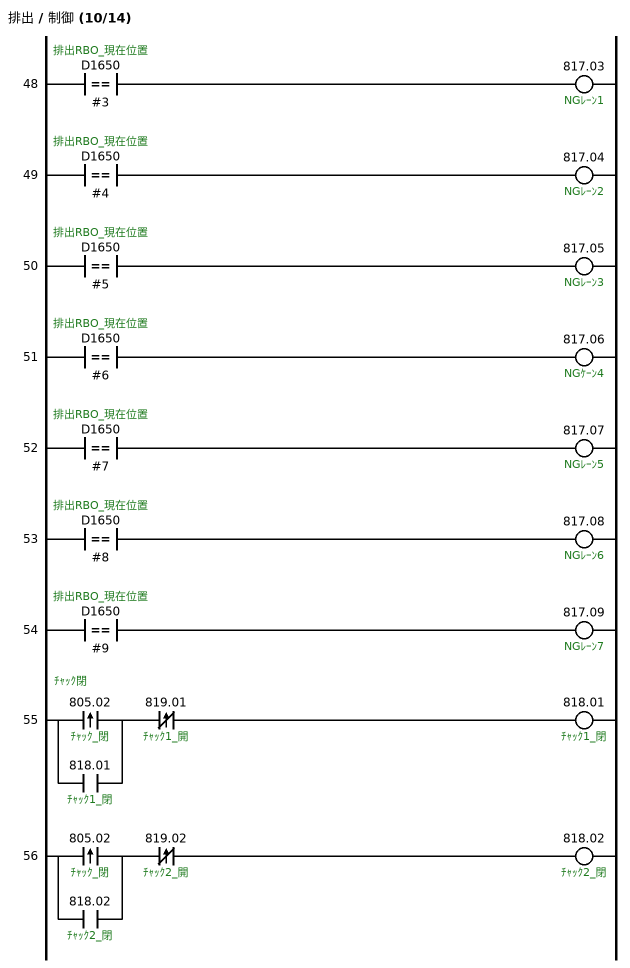
; rung 48
LD=(300) D1650 #3  ; 排出RBO_現在位置
OUT 817.03  ; NGﾚｰﾝ1
; rung 49
LD=(300) D1650 #4  ; 排出RBO_現在位置
OUT 817.04  ; NGﾚｰﾝ2
; rung 50
LD=(300) D1650 #5  ; 排出RBO_現在位置
OUT 817.05  ; NGﾚｰﾝ3
; rung 51
LD=(300) D1650 #6  ; 排出RBO_現在位置
OUT 817.06  ; NGｹｰﾝ4
; rung 52
LD=(300) D1650 #7  ; 排出RBO_現在位置
OUT 817.07  ; NGﾚｰﾝ5
; rung 53
LD=(300) D1650 #8  ; 排出RBO_現在位置
OUT 817.08  ; NGﾚｰﾝ6
; rung 54
LD=(300) D1650 #9  ; 排出RBO_現在位置
OUT 817.09  ; NGﾚｰﾝ7
; rung 55: ﾁｬｯｸ閉
@LD 805.02  ; ﾁｬｯｸ_閉
OR 818.01  ; ﾁｬｯｸ1_閉
@ANDNOT 819.01  ; ﾁｬｯｸ1_開
OUT 818.01  ; ﾁｬｯｸ1_閉
; rung 56
@LD 805.02  ; ﾁｬｯｸ_閉
OR 818.02  ; ﾁｬｯｸ2_閉
@ANDNOT 819.02  ; ﾁｬｯｸ2_開
OUT 818.02  ; ﾁｬｯｸ2_閉

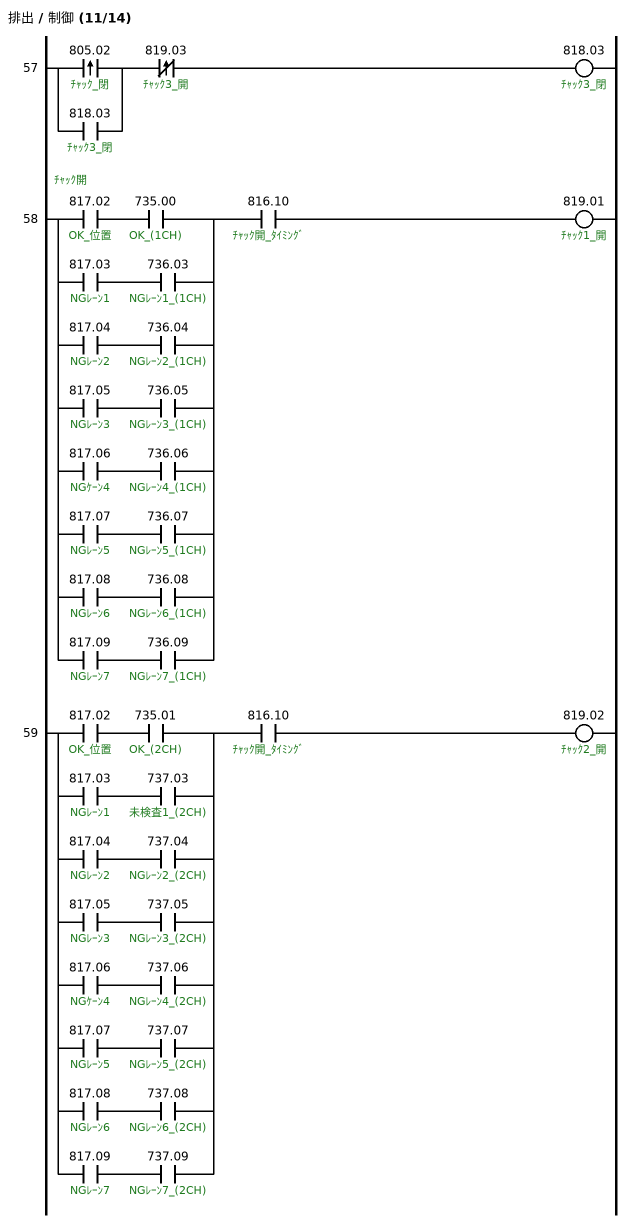
; rung 57
@LD 805.02  ; ﾁｬｯｸ_閉
OR 818.03  ; ﾁｬｯｸ3_閉
@ANDNOT 819.03  ; ﾁｬｯｸ3_開
OUT 818.03  ; ﾁｬｯｸ3_閉
; rung 58: ﾁｬｯｸ開
LD 817.02  ; OK_位置
AND 735.00  ; OK_(1CH)
LD 817.03  ; NGﾚｰﾝ1
AND 736.03  ; NGﾚｰﾝ1_(1CH)
ORLD
LD 817.04  ; NGﾚｰﾝ2
AND 736.04  ; NGﾚｰﾝ2_(1CH)
ORLD
LD 817.05  ; NGﾚｰﾝ3
AND 736.05  ; NGﾚｰﾝ3_(1CH)
ORLD
LD 817.06  ; NGｹｰﾝ4
AND 736.06  ; NGﾚｰﾝ4_(1CH)
ORLD
LD 817.07  ; NGﾚｰﾝ5
AND 736.07  ; NGﾚｰﾝ5_(1CH)
ORLD
LD 817.08  ; NGﾚｰﾝ6
AND 736.08  ; NGﾚｰﾝ6_(1CH)
ORLD
LD 817.09  ; NGﾚｰﾝ7
AND 736.09  ; NGﾚｰﾝ7_(1CH)
ORLD
AND 816.10  ; ﾁｬｯｸ開_ﾀｲﾐﾝｸﾞ
OUT 819.01  ; ﾁｬｯｸ1_開
; rung 59
LD 817.02  ; OK_位置
AND 735.01  ; OK_(2CH)
LD 817.03  ; NGﾚｰﾝ1
AND 737.03  ; 未検査1_(2CH)
ORLD
LD 817.04  ; NGﾚｰﾝ2
AND 737.04  ; NGﾚｰﾝ2_(2CH)
ORLD
LD 817.05  ; NGﾚｰﾝ3
AND 737.05  ; NGﾚｰﾝ3_(2CH)
ORLD
LD 817.06  ; NGｹｰﾝ4
AND 737.06  ; NGﾚｰﾝ4_(2CH)
ORLD
LD 817.07  ; NGﾚｰﾝ5
AND 737.07  ; NGﾚｰﾝ5_(2CH)
ORLD
LD 817.08  ; NGﾚｰﾝ6
AND 737.08  ; NGﾚｰﾝ6_(2CH)
ORLD
LD 817.09  ; NGﾚｰﾝ7
AND 737.09  ; NGﾚｰﾝ7_(2CH)
ORLD
AND 816.10  ; ﾁｬｯｸ開_ﾀｲﾐﾝｸﾞ
OUT 819.02  ; ﾁｬｯｸ2_開

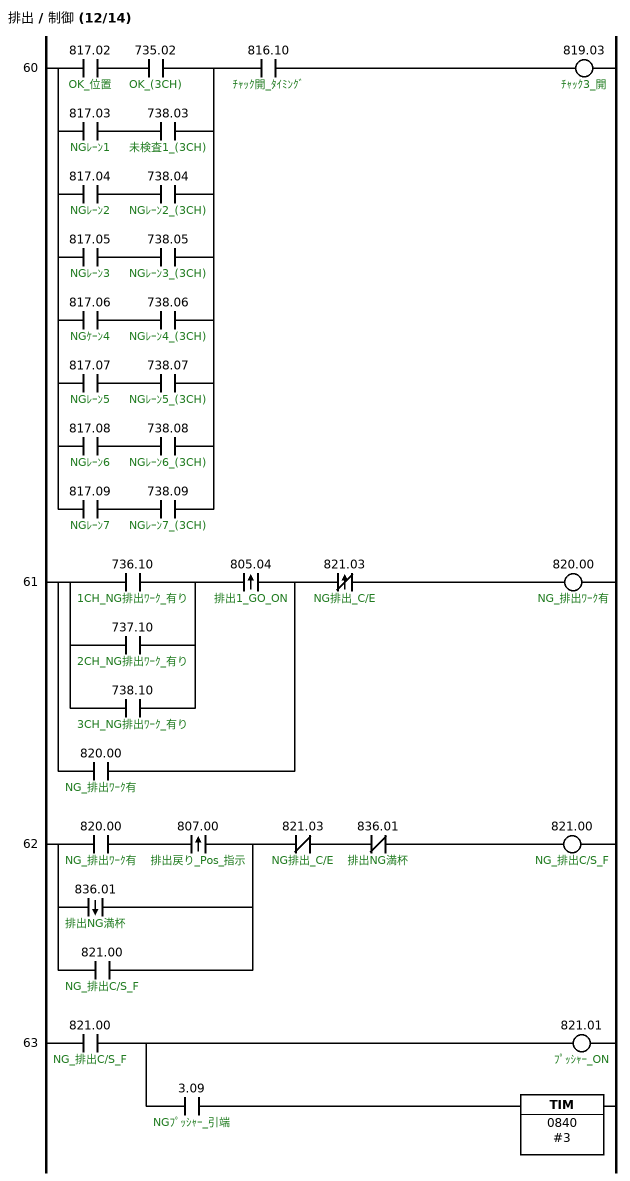
; rung 60
LD 817.02  ; OK_位置
AND 735.02  ; OK_(3CH)
LD 817.03  ; NGﾚｰﾝ1
AND 738.03  ; 未検査1_(3CH)
ORLD
LD 817.04  ; NGﾚｰﾝ2
AND 738.04  ; NGﾚｰﾝ2_(3CH)
ORLD
LD 817.05  ; NGﾚｰﾝ3
AND 738.05  ; NGﾚｰﾝ3_(3CH)
ORLD
LD 817.06  ; NGｹｰﾝ4
AND 738.06  ; NGﾚｰﾝ4_(3CH)
ORLD
LD 817.07  ; NGﾚｰﾝ5
AND 738.07  ; NGﾚｰﾝ5_(3CH)
ORLD
LD 817.08  ; NGﾚｰﾝ6
AND 738.08  ; NGﾚｰﾝ6_(3CH)
ORLD
LD 817.09  ; NGﾚｰﾝ7
AND 738.09  ; NGﾚｰﾝ7_(3CH)
ORLD
AND 816.10  ; ﾁｬｯｸ開_ﾀｲﾐﾝｸﾞ
OUT 819.03  ; ﾁｬｯｸ3_開
; rung 61
LD 736.10  ; 1CH_NG排出ﾜｰｸ_有り
OR 737.10  ; 2CH_NG排出ﾜｰｸ_有り
OR 738.10  ; 3CH_NG排出ﾜｰｸ_有り
@AND 805.04  ; 排出1_GO_ON
OR 820.00  ; NG_排出ﾜｰｸ有
@ANDNOT 821.03  ; NG排出_C/E
OUT 820.00  ; NG_排出ﾜｰｸ有
; rung 62
LD 820.00  ; NG_排出ﾜｰｸ有
@AND 807.00  ; 排出戻り_Pos_指示
%OR 836.01  ; 排出NG満杯
OR 821.00  ; NG_排出C/S_F
ANDNOT 821.03  ; NG排出_C/E
ANDNOT 836.01  ; 排出NG満杯
OUT 821.00  ; NG_排出C/S_F
; rung 63
LD 821.00  ; NG_排出C/S_F
OUT 821.01  ; ﾌﾟｯｼｬｰ_ON
AND 3.09  ; NGﾌﾟｯｼｬｰ_引端
TIM 0840 #3

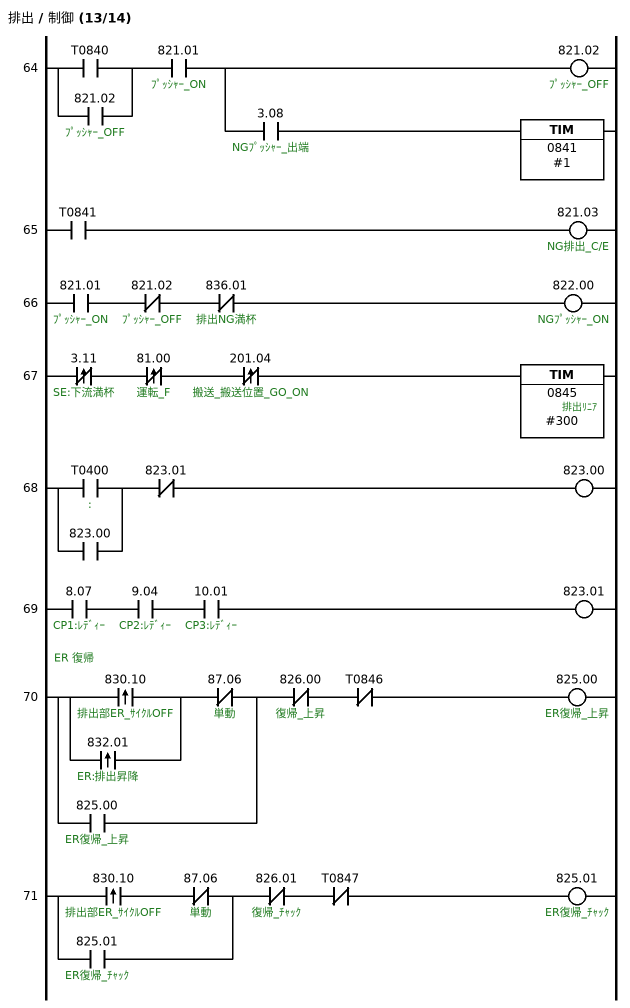
; rung 64
LD T0840
OR 821.02  ; ﾌﾟｯｼｬｰ_OFF
AND 821.01  ; ﾌﾟｯｼｬｰ_ON
OUT 821.02  ; ﾌﾟｯｼｬｰ_OFF
AND 3.08  ; NGﾌﾟｯｼｬｰ_出端
TIM 0841 #1
; rung 65
LD T0841
OUT 821.03  ; NG排出_C/E
; rung 66
LD 821.01  ; ﾌﾟｯｼｬｰ_ON
ANDNOT 821.02  ; ﾌﾟｯｼｬｰ_OFF
ANDNOT 836.01  ; 排出NG満杯
OUT 822.00  ; NGﾌﾟｯｼｬｰ_ON
; rung 67
@LDNOT 3.11  ; SE:下流満杯
@ANDNOT 81.00  ; 運転_F
@ANDNOT 201.04  ; 搬送_搬送位置_GO_ON
TIM 0845 #300  ; 排出ﾘﾆｱ
; rung 68
LD T0400  ; :
OR 823.00
ANDNOT 823.01
OUT 823.00
; rung 69
LD 8.07  ; CP1:ﾚﾃﾞｨｰ
AND 9.04  ; CP2:ﾚﾃﾞｨｰ
AND 10.01  ; CP3:ﾚﾃﾞｨｰ
OUT 823.01
; rung 70: ER 復帰
@LD 830.10  ; 排出部ER_ｻｲｸﾙOFF
@OR 832.01  ; ER:排出昇降
ANDNOT 87.06  ; 単動
OR 825.00  ; ER復帰_上昇
ANDNOT 826.00  ; 復帰_上昇
ANDNOT T0846
OUT 825.00  ; ER復帰_上昇
; rung 71
@LD 830.10  ; 排出部ER_ｻｲｸﾙOFF
ANDNOT 87.06  ; 単動
OR 825.01  ; ER復帰_ﾁｬｯｸ
ANDNOT 826.01  ; 復帰_ﾁｬｯｸ
ANDNOT T0847
OUT 825.01  ; ER復帰_ﾁｬｯｸ

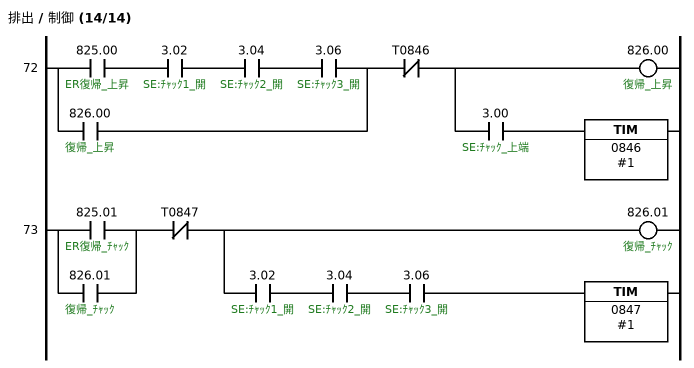
; rung 72
LD 825.00  ; ER復帰_上昇
AND 3.02  ; SE:ﾁｬｯｸ1_開
AND 3.04  ; SE:ﾁｬｯｸ2_開
AND 3.06  ; SE:ﾁｬｯｸ3_開
OR 826.00  ; 復帰_上昇
ANDNOT T0846
OUT 826.00  ; 復帰_上昇
AND 3.00  ; SE:ﾁｬｯｸ_上端
TIM 0846 #1
; rung 73
LD 825.01  ; ER復帰_ﾁｬｯｸ
OR 826.01  ; 復帰_ﾁｬｯｸ
ANDNOT T0847
OUT 826.01  ; 復帰_ﾁｬｯｸ
AND 3.02  ; SE:ﾁｬｯｸ1_開
AND 3.04  ; SE:ﾁｬｯｸ2_開
AND 3.06  ; SE:ﾁｬｯｸ3_開
TIM 0847 #1

### Section 出力

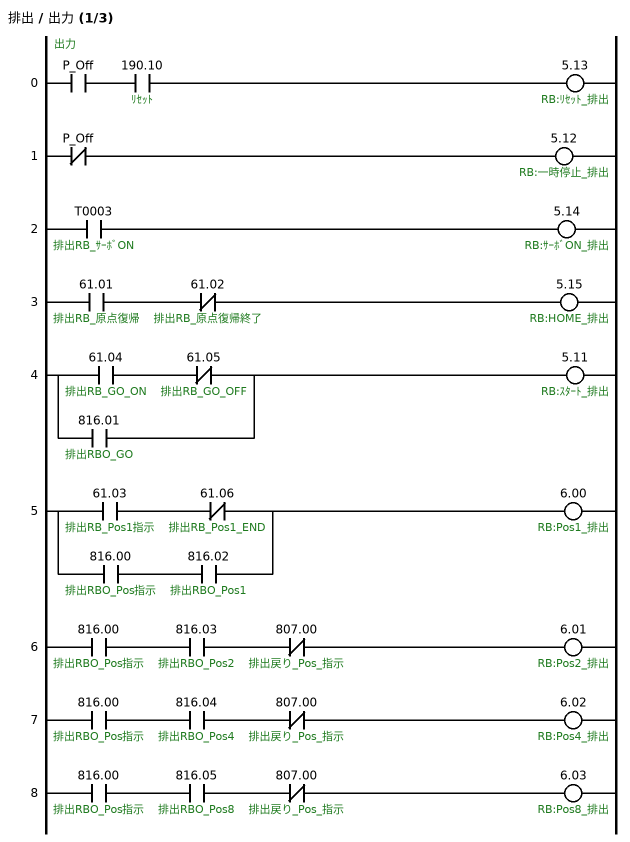
; rung 0: 出力
LD P_Off
AND 190.10  ; ﾘｾｯﾄ
OUT 5.13  ; RB:ﾘｾｯﾄ_排出
; rung 1
LDNOT P_Off
OUT 5.12  ; RB:一時停止_排出
; rung 2
LD T0003  ; 排出RB_ｻｰﾎﾞON
OUT 5.14  ; RB:ｻｰﾎﾞON_排出
; rung 3
LD 61.01  ; 排出RB_原点復帰
ANDNOT 61.02  ; 排出RB_原点復帰終了
OUT 5.15  ; RB:HOME_排出
; rung 4
LD 61.04  ; 排出RB_GO_ON
ANDNOT 61.05  ; 排出RB_GO_OFF
OR 816.01  ; 排出RBO_GO
OUT 5.11  ; RB:ｽﾀｰﾄ_排出
; rung 5
LD 61.03  ; 排出RB_Pos1指示
ANDNOT 61.06  ; 排出RB_Pos1_END
LD 816.00  ; 排出RBO_Pos指示
AND 816.02  ; 排出RBO_Pos1
ORLD
OUT 6.00  ; RB:Pos1_排出
; rung 6
LD 816.00  ; 排出RBO_Pos指示
AND 816.03  ; 排出RBO_Pos2
ANDNOT 807.00  ; 排出戻り_Pos_指示
OUT 6.01  ; RB:Pos2_排出
; rung 7
LD 816.00  ; 排出RBO_Pos指示
AND 816.04  ; 排出RBO_Pos4
ANDNOT 807.00  ; 排出戻り_Pos_指示
OUT 6.02  ; RB:Pos4_排出
; rung 8
LD 816.00  ; 排出RBO_Pos指示
AND 816.05  ; 排出RBO_Pos8
ANDNOT 807.00  ; 排出戻り_Pos_指示
OUT 6.03  ; RB:Pos8_排出

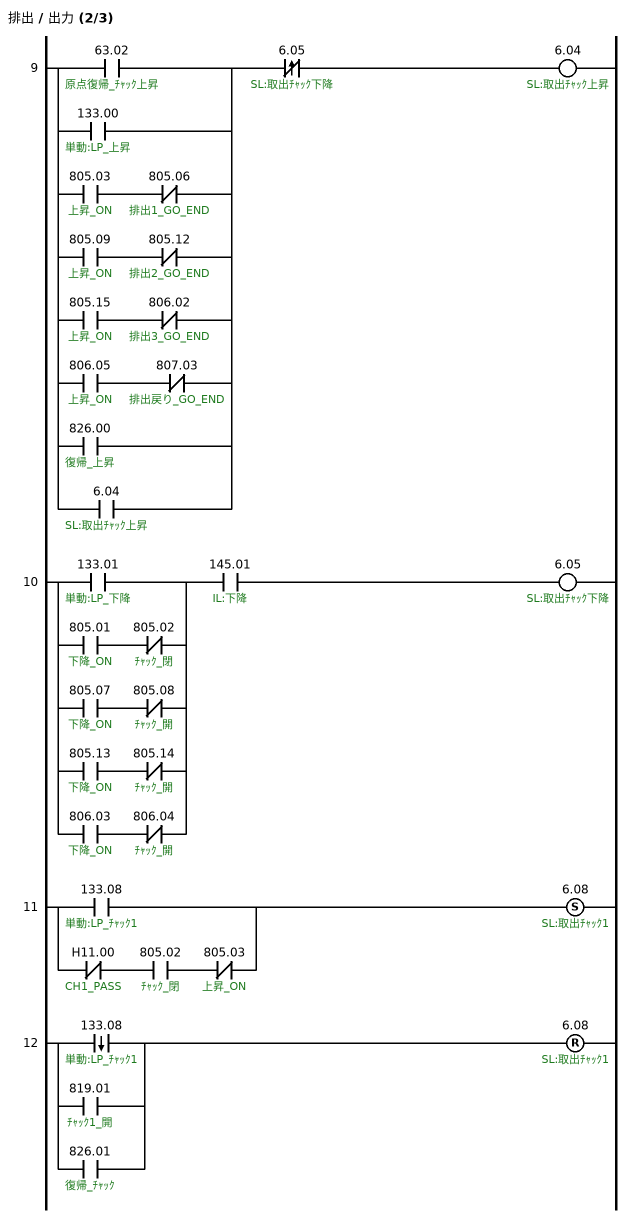
; rung 9
LD 63.02  ; 原点復帰_ﾁｬｯｸ上昇
OR 133.00  ; 単動:LP_上昇
LD 805.03  ; 上昇_ON
ANDNOT 805.06  ; 排出1_GO_END
ORLD
LD 805.09  ; 上昇_ON
ANDNOT 805.12  ; 排出2_GO_END
ORLD
LD 805.15  ; 上昇_ON
ANDNOT 806.02  ; 排出3_GO_END
ORLD
LD 806.05  ; 上昇_ON
ANDNOT 807.03  ; 排出戻り_GO_END
ORLD
OR 826.00  ; 復帰_上昇
OR 6.04  ; SL:取出ﾁｬｯｸ上昇
@ANDNOT 6.05  ; SL:取出ﾁｬｯｸ下降
OUT 6.04  ; SL:取出ﾁｬｯｸ上昇
; rung 10
LD 133.01  ; 単動:LP_下降
LD 805.01  ; 下降_ON
ANDNOT 805.02  ; ﾁｬｯｸ_閉
ORLD
LD 805.07  ; 下降_ON
ANDNOT 805.08  ; ﾁｬｯｸ_開
ORLD
LD 805.13  ; 下降_ON
ANDNOT 805.14  ; ﾁｬｯｸ_開
ORLD
LD 806.03  ; 下降_ON
ANDNOT 806.04  ; ﾁｬｯｸ_開
ORLD
AND 145.01  ; IL:下降
OUT 6.05  ; SL:取出ﾁｬｯｸ下降
; rung 11
LD 133.08  ; 単動:LP_ﾁｬｯｸ1
LDNOT H11.00  ; CH1_PASS
AND 805.02  ; ﾁｬｯｸ_閉
ANDNOT 805.03  ; 上昇_ON
ORLD
SET 6.08  ; SL:取出ﾁｬｯｸ1
; rung 12
%LD 133.08  ; 単動:LP_ﾁｬｯｸ1
OR 819.01  ; ﾁｬｯｸ1_開
OR 826.01  ; 復帰_ﾁｬｯｸ
RSET 6.08  ; SL:取出ﾁｬｯｸ1

